// TwinCAT 3 PLC project IoT_HTTP_REST_API
// ProgramVersion: 3.1.4023.0
// libraries:
//   Tc2_EtherCAT, * (Beckhoff Automation GmbH)
//   Tc2_MDP, * (Beckhoff Automation GmbH)
//   Tc2_ModbusSrv, * (Beckhoff Automation GmbH)
//   Tc2_Standard, * (Beckhoff Automation GmbH)
//   Tc2_System, * (Beckhoff Automation GmbH)
//   Tc2_Utilities, * (Beckhoff Automation GmbH)
//   Tc3_IotBase, * (Beckhoff Automation GmbH)
//   Tc3_IPCDiag, * (Beckhoff Automation GmbH)
//   Tc3_JsonXml, * (Beckhoff Automation GmbH)
//   Tc3_Module, * (Beckhoff Automation GmbH)
//   BASIC,3.31,OSCAT
//   VisuSymbols,3.5.10.0,System
// project tree:
//   / Class Diagram.TcCD (not stored), GlobalTextList.TcGTLO (not stored), PlcTask_10ms.TcTTO (not stored), PlcTask_500us.TcTTO (not stored), Task_1ms.TcTTO (not stored), Visualization Manager.TcVMO (not stored)
//   DUTs/ AirValveSimSignals.TcDUT (not stored), ElectrDataModbusTCP.TcDUT (not stored), ElectrDataEthCAT.TcDUT (not stored)
//   DUTs/DataModels/ DriveState_DataModel.TcDUT (not stored), ElectrDevicePeriodicOper_DataModel.TcDUT (not stored), ElectrDeviceContOper_DataModel.TcDUT (not stored), SingleSensor_DataModel.TcDUT (not stored), SingleState_DataModel.TcDUT (not stored), VibAccelarationDataModel.TcDUT (not stored)
//   DUTs/MES/ Order.TcDUT
//   GVLs/ GVL_const.TcGVL, GVL_SW.TcGVL (not stored), GVL_HW.TcGVL (not stored), GVL_Visu.TcGVL (not stored)
//   POUs/EL3443/EL3443/DUTs/ E_EL3443_Phase.TcDUT (not stored), E_EL3443_Total.TcDUT (not stored), ST_EL3443_MUX_REAL.TcDUT (not stored), ST_EL3443_MUX_ULINT.TcDUT (not stored), ST_EL3443_StatusLx.TcDUT (not stored), ST_EL3443_StatusTotal.TcDUT (not stored), ST_EL3443_VariantLx.TcDUT (not stored), ST_EL3443_VariantTotal.TcDUT (not stored), ST_EL3443_VariantValues.TcDUT (not stored)
//   POUs/EL3443/EL3443/ FB_EL3443.TcPOU (not stored)
//   POUs/EL3443/EL3443_DPM/DUTs/ E_EL3443_DPM_Phase.TcDUT (not stored), E_EL3443_DPM_Total.TcDUT (not stored), ST_EL3443_DPM_MUX_REAL.TcDUT (not stored), ST_EL3443_DPM_MUX_ULINT.TcDUT (not stored), ST_EL3443_DPM_StatusLx.TcDUT (not stored), ST_EL3443_DPM_StatusTotal.TcDUT (not stored), ST_EL3443_DPM_VariantLx.TcDUT (not stored), ST_EL3443_DPM_VariantTotal.TcDUT (not stored), ST_EL3443_DPM_VariantValues.TcDUT (not stored)
//   POUs/EL3443/EL3443_DPM/ FB_EL3443_DPM.TcPOU (not stored)
//   POUs/FB/Generic/ CheckLineProducing.TcPOU (not stored), PartsPerMinHistorical.TcPOU (not stored), PartsPerMinInstant.TcPOU (not stored), PartsPerMinInstant2.TcPOU (not stored), ReadMemoryUsage.TcPOU (not stored), TONR.TcPOU (not stored), UnixTimestamp.TcPOU (not stored), ValueChangeDetector.TcPOU (not stored), Valve_Signal_Sim.TcPOU (not stored)
//   POUs/FB/HTTP_REST_API/ HttpGet.TcPOU, ElectricalDevicePeriodicOper.TcPOU, ElectricalDeviceContOper.TcPOU, GenericSensor.TcPOU, GenericState.TcPOU, HttpPost.TcPOU, VibrationSensor.TcPOU
//   POUs/FB/ModbusTCP/ ReadMBSentron_PAC1200.TcPOU (not stored)
//   POUs/FC/ AI_Scale.TcPOU (not stored)
//   POUs/PRG_10ms/ PRG_06_ElectricalMonitoring.TcPOU, PRG_05_ElectricalAnalytics.TcPOU, PRG_01_MAIN.TcPOU, PRG_09_PlcDiagnostic.TcPOU, PRG_08_ProductionStatistics.TcPOU, PRG_10_TempHumidAnalytics.TcPOU, PRG_11_AirFlowAnalytics.TcPOU, PRG_12_OilContaminationAnalytics.TcPOU, PRG_13_MES.TcPOU, Simulation.TcPOU, PRG_02_DataMapping.TcPOU (not stored), PRG_07_LineState.TcPOU, PRG_03_VibrationAnalytics.TcPOU
//   POUs/PRG_1ms/ Main_T1ms.TcPOU (not stored), TimeStamp.TcPOU (not stored)
//   POUs/PRG_500us/ Main_500us.TcPOU (not stored)
//   VISU/ TextList1.TcTLO (not stored), Visualization1.TcVIS (not stored)
// real-time tasks:
//   TASK PlcTask_10ms: cycle T#10ms, priority 20, ADS port 350
//   TASK Task_1ms: cycle T#1ms, priority 1, ADS port 351
//   TASK ProfiNET: cycle T#2ms, priority 2, ADS port 301
//   TASK PlcTask_500us: cycle T#500us, priority 23, ADS port 354
// I/O:
//   DEVICE Device1 (Profinet Device) (disabled), AmsNetId 192.168.149.130.2.1
//     profinet-io-device [Beckhoff Automation TwinCAT PLC PROFINET I/O Device with I/Os, V2.32, 1 port diagnostic supported TwinCAT PN Device]
//       modules: Term 1 (DAP Module), Term 2 (32 Word Output), Term 3 (32 DWord Output), Term 4 (10 Float32 Output), Term 5 (10 Float32 Input)
//   DEVICE Device2 (EtherCAT) (disabled), AmsNetId 192.168.149.130.3.1
//     ElectricalCabinet [EK1100 EtherCAT Coupler (2A E-Bus)]
//       Term_1 (EL3443) [EL3443 3Ch. Power Measuring]
//       Term_2 (EL3443) [EL3443 3Ch. Power Measuring]
//       Term_3 (EL3152) [EL3152 2Ch. Ana Input 4-20mA]
//       Term_4 (EL6601) [EL6601 1 Port Switch (Ethernet, CoE)]
//       Term_99 (EL9011) [EL9011 End Terminal]
//     IO_LinkNode1 (EP6228-0022) [EP6228-0022 (IO Link Master)]
//       modules: Module 1 (DeviceState Inputs Device), Module 2 (DeviceState Inputs), IoLinkNode1_Ch1 (IO-Link Slave), IoLinkNode1_Ch2 (IO-Link Slave), IoLinkNode1_Ch3 (IO-Link Slave), IoLinkNode1_Ch4 (IO-Link Slave), IoLinkNode1_Ch5 (IO-Link Slave), IoLinkNode1_Ch6 (IO-Link Slave), Module 9 (empty), Module 10 (empty)
//     IO_LinkNode2 (EP6224-2022) [EP6224-2022 (IO Link Master)]
//       modules: Module 1 (DeviceState Inputs Device), Module 2 (DeviceState Inputs), IoLinkNode2_Ch1 (IO-Link Slave), IoLinkNode2_Ch2 (IO-Link Slave), IoLinkNode2_Ch3 (IO-Link Slave), IoLinkNode2_Ch4 (IO-Link Slave)
//   DEVICE Device 3 (USB) (disabled)
//     Box 2 (C9900-L100 License-Key-USB-Stick)
// variable links:
//   IoT_HTTP_REST_API/IoT_HTTP_REST_API Instance <-> Device1 (Profinet Device)/profinet-io-device
//     PlcTask_10ms Inputs/GVL_HW.PnIoDevice_10Real_In <-> API/Term 4 (10 Float32 Output)/Subterm 6 (10 Float32 Output)/Inputs/1 Float32 Output[0]
//     PlcTask_10ms Inputs/GVL_HW.PnIoDevice_10Real_In @bit {32..288 step 32} <-> API/Term 4 (10 Float32 Output)/Subterm 6 (10 Float32 Output)/Inputs/1 Float32 Output[{1..9}]  (9 links)
//     PlcTask_10ms Inputs/GVL_HW.PnIoDevice_32DWord_In <-> API/Term 3 (32 DWord Output)/Subterm 5 (32 DWord Output)/Inputs/1 DWord Output[0]
//     PlcTask_10ms Inputs/GVL_HW.PnIoDevice_32DWord_In @bit {32..992 step 32} <-> API/Term 3 (32 DWord Output)/Subterm 5 (32 DWord Output)/Inputs/1 DWord Output[{1..31}]  (31 links)
//     PlcTask_10ms Inputs/GVL_HW.PnIoDevice_32Word_In <-> API/Term 2 (32 Word Output)/Subterm 4 (32 Word Output)/Inputs/1 Word Output[0]
//     PlcTask_10ms Inputs/GVL_HW.PnIoDevice_32Word_In @bit {16..496 step 16} <-> API/Term 2 (32 Word Output)/Subterm 4 (32 Word Output)/Inputs/1 Word Output[{1..31}]  (31 links)
//     PlcTask_10ms Outputs/GVL_HW.PnIoDevice_10Real_Out <-> API/Term 5 (10 Float32 Input)/Subterm 7 (10 Float32 Input)/Outputs/1 Float32 Input[0]
//     PlcTask_10ms Outputs/GVL_HW.PnIoDevice_10Real_Out @bit {32..288 step 32} <-> API/Term 5 (10 Float32 Input)/Subterm 7 (10 Float32 Input)/Outputs/1 Float32 Input[{1..9}]  (9 links)
//   IoT_HTTP_REST_API/IoT_HTTP_REST_API Instance <-> Device2 (EtherCAT)/ElectricalCabinet/Term_1 (EL3443)
//     PlcTask_500us Inputs/Main_500us.ElectricalDevice1.stEL3443_IO.MDP5001_341_Input/MDP5001_341_L1_Basic_Current <-> L1 Basic/Current
//     PlcTask_500us Inputs/Main_500us.ElectricalDevice1.stEL3443_IO.MDP5001_341_Input/MDP5001_341_L2_Basic_Current <-> L2 Basic/Current
//     PlcTask_500us Inputs/Main_500us.ElectricalDevice1.stEL3443_IO.MDP5001_341_Input/MDP5001_341_L3_Basic_Current <-> L3 Basic/Current
//     PlcTask_500us Inputs/Main_500us.ElectricalDevice1.stEL3443_IO.MDP5001_341_Input/MDP5001_341_L1_Basic_Voltage <-> L1 Basic/Voltage
//     PlcTask_500us Inputs/Main_500us.ElectricalDevice1.stEL3443_IO.MDP5001_341_Input/MDP5001_341_L2_Basic_Voltage <-> L2 Basic/Voltage
//     PlcTask_500us Inputs/Main_500us.ElectricalDevice1.stEL3443_IO.MDP5001_341_Input/MDP5001_341_L3_Basic_Voltage <-> L3 Basic/Voltage
//     PlcTask_500us Inputs/Main_500us.ElectricalDevice1.stEL3443_IO.MDP5001_341_Input/MDP5001_341_L1_Power_Active_Power <-> L1 Power/Active Power
//     PlcTask_500us Inputs/Main_500us.ElectricalDevice1.stEL3443_IO.MDP5001_341_Input/MDP5001_341_L2_Power_Active_Power <-> L2 Power/Active Power
//     PlcTask_500us Inputs/Main_500us.ElectricalDevice1.stEL3443_IO.MDP5001_341_Input/MDP5001_341_L3_Power_Active_Power <-> L3 Power/Active Power
//     PlcTask_500us Inputs/Main_500us.ElectricalDevice1.stEL3443_IO.MDP5001_341_Input/MDP5001_341_L1_Power_Apparent_Power <-> L1 Power/Apparent Power
//     PlcTask_500us Inputs/Main_500us.ElectricalDevice1.stEL3443_IO.MDP5001_341_Input/MDP5001_341_L2_Power_Apparent_Power <-> L2 Power/Apparent Power
//     PlcTask_500us Inputs/Main_500us.ElectricalDevice1.stEL3443_IO.MDP5001_341_Input/MDP5001_341_L3_Power_Apparent_Power <-> L3 Power/Apparent Power
//     PlcTask_500us Inputs/Main_500us.ElectricalDevice1.stEL3443_IO.MDP5001_341_Input/MDP5001_341_L1_Power_Power_Factor <-> L1 Power/Power Factor
//     PlcTask_500us Inputs/Main_500us.ElectricalDevice1.stEL3443_IO.MDP5001_341_Input/MDP5001_341_L2_Power_Power_Factor <-> L2 Power/Power Factor
//     PlcTask_500us Inputs/Main_500us.ElectricalDevice1.stEL3443_IO.MDP5001_341_Input/MDP5001_341_L3_Power_Power_Factor <-> L3 Power/Power Factor
//     PlcTask_500us Inputs/Main_500us.ElectricalDevice1.stEL3443_IO.MDP5001_341_Input/MDP5001_341_L1_Power_Reactive_Power <-> L1 Power/Reactive Power
//     PlcTask_500us Inputs/Main_500us.ElectricalDevice1.stEL3443_IO.MDP5001_341_Input/MDP5001_341_L2_Power_Reactive_Power <-> L2 Power/Reactive Power
//     PlcTask_500us Inputs/Main_500us.ElectricalDevice1.stEL3443_IO.MDP5001_341_Input/MDP5001_341_L3_Power_Reactive_Power <-> L3 Power/Reactive Power
//     PlcTask_500us Inputs/Main_500us.ElectricalDevice1.stEL3443_IO.MDP5001_341_Input/MDP5001_341_L1_Status_Current_Guard_Error <-> L1 Status/Current Guard Error
//     PlcTask_500us Inputs/Main_500us.ElectricalDevice1.stEL3443_IO.MDP5001_341_Input/MDP5001_341_L2_Status_Current_Guard_Error <-> L2 Status/Current Guard Error
//     PlcTask_500us Inputs/Main_500us.ElectricalDevice1.stEL3443_IO.MDP5001_341_Input/MDP5001_341_L3_Status_Current_Guard_Error <-> L3 Status/Current Guard Error
//     PlcTask_500us Inputs/Main_500us.ElectricalDevice1.stEL3443_IO.MDP5001_341_Input/MDP5001_341_L1_Status_Current_Guard_Warning <-> L1 Status/Current Guard Warning
//     PlcTask_500us Inputs/Main_500us.ElectricalDevice1.stEL3443_IO.MDP5001_341_Input/MDP5001_341_L2_Status_Current_Guard_Warning <-> L2 Status/Current Guard Warning
//     PlcTask_500us Inputs/Main_500us.ElectricalDevice1.stEL3443_IO.MDP5001_341_Input/MDP5001_341_L3_Status_Current_Guard_Warning <-> L3 Status/Current Guard Warning
//     PlcTask_500us Inputs/Main_500us.ElectricalDevice1.stEL3443_IO.MDP5001_341_Input/MDP5001_341_L1_Status_Inaccurate_Current <-> L1 Status/Inaccurate Current
//     PlcTask_500us Inputs/Main_500us.ElectricalDevice1.stEL3443_IO.MDP5001_341_Input/MDP5001_341_L2_Status_Inaccurate_Current <-> L2 Status/Inaccurate Current
//     PlcTask_500us Inputs/Main_500us.ElectricalDevice1.stEL3443_IO.MDP5001_341_Input/MDP5001_341_L3_Status_Inaccurate_Current <-> L3 Status/Inaccurate Current
//     PlcTask_500us Inputs/Main_500us.ElectricalDevice1.stEL3443_IO.MDP5001_341_Input/MDP5001_341_L1_Status_Inaccurate_Voltage <-> L1 Status/Inaccurate Voltage
//     PlcTask_500us Inputs/Main_500us.ElectricalDevice1.stEL3443_IO.MDP5001_341_Input/MDP5001_341_L2_Status_Inaccurate_Voltage <-> L2 Status/Inaccurate Voltage
//     PlcTask_500us Inputs/Main_500us.ElectricalDevice1.stEL3443_IO.MDP5001_341_Input/MDP5001_341_L3_Status_Inaccurate_Voltage <-> L3 Status/Inaccurate Voltage
//     PlcTask_500us Inputs/Main_500us.ElectricalDevice1.stEL3443_IO.MDP5001_341_Input/MDP5001_341_L1_Status_Overcurrent <-> L1 Status/Overcurrent
//     PlcTask_500us Inputs/Main_500us.ElectricalDevice1.stEL3443_IO.MDP5001_341_Input/MDP5001_341_L2_Status_Overcurrent <-> L2 Status/Overcurrent
//     PlcTask_500us Inputs/Main_500us.ElectricalDevice1.stEL3443_IO.MDP5001_341_Input/MDP5001_341_L3_Status_Overcurrent <-> L3 Status/Overcurrent
//     PlcTask_500us Inputs/Main_500us.ElectricalDevice1.stEL3443_IO.MDP5001_341_Input/MDP5001_341_L1_Status_Overvoltage <-> L1 Status/Overvoltage
//     PlcTask_500us Inputs/Main_500us.ElectricalDevice1.stEL3443_IO.MDP5001_341_Input/MDP5001_341_L2_Status_Overvoltage <-> L2 Status/Overvoltage
//     PlcTask_500us Inputs/Main_500us.ElectricalDevice1.stEL3443_IO.MDP5001_341_Input/MDP5001_341_L3_Status_Overvoltage <-> L3 Status/Overvoltage
//     PlcTask_500us Inputs/Main_500us.ElectricalDevice1.stEL3443_IO.MDP5001_341_Input/MDP5001_341_L1_Status_TxPDO_Toggle <-> L1 Status/TxPDO Toggle
//     PlcTask_500us Inputs/Main_500us.ElectricalDevice1.stEL3443_IO.MDP5001_341_Input/MDP5001_341_L2_Status_TxPDO_Toggle <-> L2 Status/TxPDO Toggle
//     PlcTask_500us Inputs/Main_500us.ElectricalDevice1.stEL3443_IO.MDP5001_341_Input/MDP5001_341_L3_Status_TxPDO_Toggle <-> L3 Status/TxPDO Toggle
//     PlcTask_500us Inputs/Main_500us.ElectricalDevice1.stEL3443_IO.MDP5001_341_Input/MDP5001_341_L1_Status_Voltage_Guard_Error <-> L1 Status/Voltage Guard Error
//     PlcTask_500us Inputs/Main_500us.ElectricalDevice1.stEL3443_IO.MDP5001_341_Input/MDP5001_341_L2_Status_Voltage_Guard_Error <-> L2 Status/Voltage Guard Error
//     PlcTask_500us Inputs/Main_500us.ElectricalDevice1.stEL3443_IO.MDP5001_341_Input/MDP5001_341_L3_Status_Voltage_Guard_Error <-> L3 Status/Voltage Guard Error
//     PlcTask_500us Inputs/Main_500us.ElectricalDevice1.stEL3443_IO.MDP5001_341_Input/MDP5001_341_L1_Status_Voltage_Guard_Warning <-> L1 Status/Voltage Guard Warning
//     PlcTask_500us Inputs/Main_500us.ElectricalDevice1.stEL3443_IO.MDP5001_341_Input/MDP5001_341_L2_Status_Voltage_Guard_Warning <-> L2 Status/Voltage Guard Warning
//     PlcTask_500us Inputs/Main_500us.ElectricalDevice1.stEL3443_IO.MDP5001_341_Input/MDP5001_341_L3_Status_Voltage_Guard_Warning <-> L3 Status/Voltage Guard Warning
//     PlcTask_500us Inputs/Main_500us.ElectricalDevice1.stEL3443_IO.MDP5001_341_Input/MDP5001_341_L1_Status_Voltage_Sign_Bit <-> L1 Status/Voltage Sign Bit
//     PlcTask_500us Inputs/Main_500us.ElectricalDevice1.stEL3443_IO.MDP5001_341_Input/MDP5001_341_L2_Status_Voltage_Sign_Bit <-> L2 Status/Voltage Sign Bit
//     PlcTask_500us Inputs/Main_500us.ElectricalDevice1.stEL3443_IO.MDP5001_341_Input/MDP5001_341_L3_Status_Voltage_Sign_Bit <-> L3 Status/Voltage Sign Bit
//     PlcTask_500us Inputs/Main_500us.ElectricalDevice1.stEL3443_IO.MDP5001_341_Input/MDP5001_341_L1_Timing_Voltage_Last_Zero_Crossing <-> L1 Timing/Voltage Last Zero Crossing
//     PlcTask_500us Inputs/Main_500us.ElectricalDevice1.stEL3443_IO.MDP5001_341_Input/MDP5001_341_L2_Timing_Voltage_Last_Zero_Crossing <-> L2 Timing/Voltage Last Zero Crossing
//     PlcTask_500us Inputs/Main_500us.ElectricalDevice1.stEL3443_IO.MDP5001_341_Input/MDP5001_341_L3_Timing_Voltage_Last_Zero_Crossing <-> L3 Timing/Voltage Last Zero Crossing
//     PlcTask_500us Inputs/Main_500us.ElectricalDevice1.stEL3443_IO.MDP5001_341_Input/MDP5001_341_Total_Basic_Calculated_Neutral_Line_Current <-> Total Basic/Calculated Neutral Line Current
//     PlcTask_500us Inputs/Main_500us.ElectricalDevice1.stEL3443_IO.MDP5001_341_Input/MDP5001_341_Total_Basic_Frequency <-> Total Basic/Frequency
//     PlcTask_500us Inputs/Main_500us.ElectricalDevice1.stEL3443_IO.MDP5001_341_Input/MDP5001_341_Total_Basic_Power_Factor <-> Total Basic/Power Factor
//     PlcTask_500us Inputs/Main_500us.ElectricalDevice1.stEL3443_IO.MDP5001_341_Input/MDP5001_341_Total_Status_Active_Power_Guard_Error <-> Total Status/Active Power Guard Error
//     PlcTask_500us Inputs/Main_500us.ElectricalDevice1.stEL3443_IO.MDP5001_341_Input/MDP5001_341_Total_Status_Active_Power_Guard_Warning <-> Total Status/Active Power Guard Warning
//     PlcTask_500us Inputs/Main_500us.ElectricalDevice1.stEL3443_IO.MDP5001_341_Input/MDP5001_341_Total_Status_Apparent_Power_Guard_Error <-> Total Status/Apparent Power Guard Error
//     PlcTask_500us Inputs/Main_500us.ElectricalDevice1.stEL3443_IO.MDP5001_341_Input/MDP5001_341_Total_Status_Apparent_Power_Guard_Warning <-> Total Status/Apparent Power Guard Warning
//     PlcTask_500us Inputs/Main_500us.ElectricalDevice1.stEL3443_IO.MDP5001_341_Input/MDP5001_341_Total_Status_Frequency_Guard_Error <-> Total Status/Frequency Guard Error
//     PlcTask_500us Inputs/Main_500us.ElectricalDevice1.stEL3443_IO.MDP5001_341_Input/MDP5001_341_Total_Status_Frequency_Guard_Warning <-> Total Status/Frequency Guard Warning
//     PlcTask_500us Inputs/Main_500us.ElectricalDevice1.stEL3443_IO.MDP5001_341_Input/MDP5001_341_Total_Status_Grid_Direction <-> Total Status/Grid Direction
//     PlcTask_500us Inputs/Main_500us.ElectricalDevice1.stEL3443_IO.MDP5001_341_Input/MDP5001_341_Total_Status_Neutral_Current_Guard_Error <-> Total Status/Neutral Current Guard Error
//     PlcTask_500us Inputs/Main_500us.ElectricalDevice1.stEL3443_IO.MDP5001_341_Input/MDP5001_341_Total_Status_Neutral_Current_Guard_Warning <-> Total Status/Neutral Current Guard Warning
//     PlcTask_500us Inputs/Main_500us.ElectricalDevice1.stEL3443_IO.MDP5001_341_Input/MDP5001_341_Total_Status_Power_Quality_Factor <-> Total Status/Power Quality Factor
//     PlcTask_500us Inputs/Main_500us.ElectricalDevice1.stEL3443_IO.MDP5001_341_Input/MDP5001_341_Total_Status_Power_Quality_Guard_Error <-> Total Status/Power Quality Guard Error
//     PlcTask_500us Inputs/Main_500us.ElectricalDevice1.stEL3443_IO.MDP5001_341_Input/MDP5001_341_Total_Status_Power_Quality_Guard_Warning <-> Total Status/Power Quality Guard Warning
//     PlcTask_500us Inputs/Main_500us.ElectricalDevice1.stEL3443_IO.MDP5001_341_Input/MDP5001_341_Total_Status_System_State <-> Total Status/System State
//     PlcTask_500us Inputs/Main_500us.ElectricalDevice1.stEL3443_IO.MDP5001_341_Input/MDP5001_341_Total_Status_TxPDO_State <-> Total Status/TxPDO State
//     PlcTask_500us Inputs/Main_500us.ElectricalDevice1.stEL3443_IO.MDP5001_341_Input/MDP5001_341_Total_Status_TxPDO_Toggle <-> Total Status/TxPDO Toggle
//     PlcTask_500us Inputs/Main_500us.ElectricalDevice1.stEL3443_IO.MDP5001_341_Input/MDP5001_341_Total_Variant_Value_In_Index_1_REAL <-> Total Variant Value In/Index 1 REAL
//     PlcTask_500us Inputs/Main_500us.ElectricalDevice1.stEL3443_IO.MDP5001_341_Input/MDP5001_341_Total_Variant_Value_In_Index_2_REAL <-> Total Variant Value In/Index 2 REAL
//     PlcTask_500us Inputs/Main_500us.ElectricalDevice1.stEL3443_IO.MDP5001_341_Input/MDP5001_341_Total_Variant_Value_In_Index_3_REAL <-> Total Variant Value In/Index 3 REAL
//     PlcTask_500us Inputs/Main_500us.ElectricalDevice1.stEL3443_IO.MDP5001_341_Input/MDP5001_341_Total_Variant_Value_In_Index_4_ULINT <-> Total Variant Value In/Index 4 ULINT
//     PlcTask_500us Inputs/Main_500us.ElectricalDevice1.stEL3443_IO.MDP5001_341_Input/MDP5001_341_Total_Variant_Value_In_TxPDO_Toggle <-> Total Variant Value In/TxPDO Toggle
//     PlcTask_500us Inputs/Main_500us.ElectricalDevice1.stEL3443_IO.MDP5001_341_Input/MDP5001_341_Total_Variant_Value_In_Value_1_REAL <-> Total Variant Value In/Value 1 REAL
//     PlcTask_500us Inputs/Main_500us.ElectricalDevice1.stEL3443_IO.MDP5001_341_Input/MDP5001_341_Total_Variant_Value_In_Value_2_REAL <-> Total Variant Value In/Value 2 REAL
//     PlcTask_500us Inputs/Main_500us.ElectricalDevice1.stEL3443_IO.MDP5001_341_Input/MDP5001_341_Total_Variant_Value_In_Value_3_REAL <-> Total Variant Value In/Value 3 REAL
//     PlcTask_500us Inputs/Main_500us.ElectricalDevice1.stEL3443_IO.MDP5001_341_Input/MDP5001_341_Total_Variant_Value_In_Value_4_ULINT <-> Total Variant Value In/Value 4 ULINT
//     PlcTask_500us Outputs/Main_500us.ElectricalDevice1.stEL3443_IO.MDP5001_341_Output/MDP5001_341_Total_Variant_Value_Out_Index_1_REAL <-> Total Variant Value Out/Index 1 REAL
//     PlcTask_500us Outputs/Main_500us.ElectricalDevice1.stEL3443_IO.MDP5001_341_Output/MDP5001_341_Total_Variant_Value_Out_Index_2_REAL <-> Total Variant Value Out/Index 2 REAL
//     PlcTask_500us Outputs/Main_500us.ElectricalDevice1.stEL3443_IO.MDP5001_341_Output/MDP5001_341_Total_Variant_Value_Out_Index_3_REAL <-> Total Variant Value Out/Index 3 REAL
//     PlcTask_500us Outputs/Main_500us.ElectricalDevice1.stEL3443_IO.MDP5001_341_Output/MDP5001_341_Total_Variant_Value_Out_Index_4_ULINT <-> Total Variant Value Out/Index 4 ULINT
//   IoT_HTTP_REST_API/IoT_HTTP_REST_API Instance <-> Device2 (EtherCAT)/ElectricalCabinet/Term_2 (EL3443)
//     PlcTask_500us Inputs/Main_500us.ElectricalDevice2.stEL3443_IO.MDP5001_341_Input/MDP5001_341_L1_Basic_Current <-> L1 Basic/Current
//     PlcTask_500us Inputs/Main_500us.ElectricalDevice2.stEL3443_IO.MDP5001_341_Input/MDP5001_341_L2_Basic_Current <-> L2 Basic/Current
//     PlcTask_500us Inputs/Main_500us.ElectricalDevice2.stEL3443_IO.MDP5001_341_Input/MDP5001_341_L3_Basic_Current <-> L3 Basic/Current
//     PlcTask_500us Inputs/Main_500us.ElectricalDevice2.stEL3443_IO.MDP5001_341_Input/MDP5001_341_L1_Basic_Voltage <-> L1 Basic/Voltage
//     PlcTask_500us Inputs/Main_500us.ElectricalDevice2.stEL3443_IO.MDP5001_341_Input/MDP5001_341_L2_Basic_Voltage <-> L2 Basic/Voltage
//     PlcTask_500us Inputs/Main_500us.ElectricalDevice2.stEL3443_IO.MDP5001_341_Input/MDP5001_341_L3_Basic_Voltage <-> L3 Basic/Voltage
//     PlcTask_500us Inputs/Main_500us.ElectricalDevice2.stEL3443_IO.MDP5001_341_Input/MDP5001_341_L1_Power_Active_Power <-> L1 Power/Active Power
//     PlcTask_500us Inputs/Main_500us.ElectricalDevice2.stEL3443_IO.MDP5001_341_Input/MDP5001_341_L2_Power_Active_Power <-> L2 Power/Active Power
//     PlcTask_500us Inputs/Main_500us.ElectricalDevice2.stEL3443_IO.MDP5001_341_Input/MDP5001_341_L3_Power_Active_Power <-> L3 Power/Active Power
//     PlcTask_500us Inputs/Main_500us.ElectricalDevice2.stEL3443_IO.MDP5001_341_Input/MDP5001_341_L1_Power_Apparent_Power <-> L1 Power/Apparent Power
//     PlcTask_500us Inputs/Main_500us.ElectricalDevice2.stEL3443_IO.MDP5001_341_Input/MDP5001_341_L2_Power_Apparent_Power <-> L2 Power/Apparent Power
//     PlcTask_500us Inputs/Main_500us.ElectricalDevice2.stEL3443_IO.MDP5001_341_Input/MDP5001_341_L3_Power_Apparent_Power <-> L3 Power/Apparent Power
//     PlcTask_500us Inputs/Main_500us.ElectricalDevice2.stEL3443_IO.MDP5001_341_Input/MDP5001_341_L1_Power_Power_Factor <-> L1 Power/Power Factor
//     PlcTask_500us Inputs/Main_500us.ElectricalDevice2.stEL3443_IO.MDP5001_341_Input/MDP5001_341_L2_Power_Power_Factor <-> L2 Power/Power Factor
//     PlcTask_500us Inputs/Main_500us.ElectricalDevice2.stEL3443_IO.MDP5001_341_Input/MDP5001_341_L3_Power_Power_Factor <-> L3 Power/Power Factor
//     PlcTask_500us Inputs/Main_500us.ElectricalDevice2.stEL3443_IO.MDP5001_341_Input/MDP5001_341_L1_Power_Reactive_Power <-> L1 Power/Reactive Power
//     PlcTask_500us Inputs/Main_500us.ElectricalDevice2.stEL3443_IO.MDP5001_341_Input/MDP5001_341_L2_Power_Reactive_Power <-> L2 Power/Reactive Power
//     PlcTask_500us Inputs/Main_500us.ElectricalDevice2.stEL3443_IO.MDP5001_341_Input/MDP5001_341_L3_Power_Reactive_Power <-> L3 Power/Reactive Power
//     PlcTask_500us Inputs/Main_500us.ElectricalDevice2.stEL3443_IO.MDP5001_341_Input/MDP5001_341_L1_Status_Current_Guard_Error <-> L1 Status/Current Guard Error
//     PlcTask_500us Inputs/Main_500us.ElectricalDevice2.stEL3443_IO.MDP5001_341_Input/MDP5001_341_L2_Status_Current_Guard_Error <-> L2 Status/Current Guard Error
//     PlcTask_500us Inputs/Main_500us.ElectricalDevice2.stEL3443_IO.MDP5001_341_Input/MDP5001_341_L3_Status_Current_Guard_Error <-> L3 Status/Current Guard Error
//     PlcTask_500us Inputs/Main_500us.ElectricalDevice2.stEL3443_IO.MDP5001_341_Input/MDP5001_341_L1_Status_Current_Guard_Warning <-> L1 Status/Current Guard Warning
//     PlcTask_500us Inputs/Main_500us.ElectricalDevice2.stEL3443_IO.MDP5001_341_Input/MDP5001_341_L2_Status_Current_Guard_Warning <-> L2 Status/Current Guard Warning
//     PlcTask_500us Inputs/Main_500us.ElectricalDevice2.stEL3443_IO.MDP5001_341_Input/MDP5001_341_L3_Status_Current_Guard_Warning <-> L3 Status/Current Guard Warning
//     PlcTask_500us Inputs/Main_500us.ElectricalDevice2.stEL3443_IO.MDP5001_341_Input/MDP5001_341_L1_Status_Inaccurate_Current <-> L1 Status/Inaccurate Current
//     PlcTask_500us Inputs/Main_500us.ElectricalDevice2.stEL3443_IO.MDP5001_341_Input/MDP5001_341_L2_Status_Inaccurate_Current <-> L2 Status/Inaccurate Current
//     PlcTask_500us Inputs/Main_500us.ElectricalDevice2.stEL3443_IO.MDP5001_341_Input/MDP5001_341_L3_Status_Inaccurate_Current <-> L3 Status/Inaccurate Current
//     PlcTask_500us Inputs/Main_500us.ElectricalDevice2.stEL3443_IO.MDP5001_341_Input/MDP5001_341_L1_Status_Inaccurate_Voltage <-> L1 Status/Inaccurate Voltage
//     PlcTask_500us Inputs/Main_500us.ElectricalDevice2.stEL3443_IO.MDP5001_341_Input/MDP5001_341_L2_Status_Inaccurate_Voltage <-> L2 Status/Inaccurate Voltage
//     PlcTask_500us Inputs/Main_500us.ElectricalDevice2.stEL3443_IO.MDP5001_341_Input/MDP5001_341_L3_Status_Inaccurate_Voltage <-> L3 Status/Inaccurate Voltage
//     PlcTask_500us Inputs/Main_500us.ElectricalDevice2.stEL3443_IO.MDP5001_341_Input/MDP5001_341_L1_Status_Overcurrent <-> L1 Status/Overcurrent
//     PlcTask_500us Inputs/Main_500us.ElectricalDevice2.stEL3443_IO.MDP5001_341_Input/MDP5001_341_L2_Status_Overcurrent <-> L2 Status/Overcurrent
//     PlcTask_500us Inputs/Main_500us.ElectricalDevice2.stEL3443_IO.MDP5001_341_Input/MDP5001_341_L3_Status_Overcurrent <-> L3 Status/Overcurrent
//     PlcTask_500us Inputs/Main_500us.ElectricalDevice2.stEL3443_IO.MDP5001_341_Input/MDP5001_341_L1_Status_Overvoltage <-> L1 Status/Overvoltage
//     PlcTask_500us Inputs/Main_500us.ElectricalDevice2.stEL3443_IO.MDP5001_341_Input/MDP5001_341_L2_Status_Overvoltage <-> L2 Status/Overvoltage
//     PlcTask_500us Inputs/Main_500us.ElectricalDevice2.stEL3443_IO.MDP5001_341_Input/MDP5001_341_L3_Status_Overvoltage <-> L3 Status/Overvoltage
//     PlcTask_500us Inputs/Main_500us.ElectricalDevice2.stEL3443_IO.MDP5001_341_Input/MDP5001_341_L1_Status_TxPDO_Toggle <-> L1 Status/TxPDO Toggle
//     PlcTask_500us Inputs/Main_500us.ElectricalDevice2.stEL3443_IO.MDP5001_341_Input/MDP5001_341_L2_Status_TxPDO_Toggle <-> L2 Status/TxPDO Toggle
//     PlcTask_500us Inputs/Main_500us.ElectricalDevice2.stEL3443_IO.MDP5001_341_Input/MDP5001_341_L3_Status_TxPDO_Toggle <-> L3 Status/TxPDO Toggle
//     PlcTask_500us Inputs/Main_500us.ElectricalDevice2.stEL3443_IO.MDP5001_341_Input/MDP5001_341_L1_Status_Voltage_Guard_Error <-> L1 Status/Voltage Guard Error
//     PlcTask_500us Inputs/Main_500us.ElectricalDevice2.stEL3443_IO.MDP5001_341_Input/MDP5001_341_L2_Status_Voltage_Guard_Error <-> L2 Status/Voltage Guard Error
//     PlcTask_500us Inputs/Main_500us.ElectricalDevice2.stEL3443_IO.MDP5001_341_Input/MDP5001_341_L3_Status_Voltage_Guard_Error <-> L3 Status/Voltage Guard Error
//     PlcTask_500us Inputs/Main_500us.ElectricalDevice2.stEL3443_IO.MDP5001_341_Input/MDP5001_341_L1_Status_Voltage_Guard_Warning <-> L1 Status/Voltage Guard Warning
//     PlcTask_500us Inputs/Main_500us.ElectricalDevice2.stEL3443_IO.MDP5001_341_Input/MDP5001_341_L2_Status_Voltage_Guard_Warning <-> L2 Status/Voltage Guard Warning
//     PlcTask_500us Inputs/Main_500us.ElectricalDevice2.stEL3443_IO.MDP5001_341_Input/MDP5001_341_L3_Status_Voltage_Guard_Warning <-> L3 Status/Voltage Guard Warning
//     PlcTask_500us Inputs/Main_500us.ElectricalDevice2.stEL3443_IO.MDP5001_341_Input/MDP5001_341_L1_Status_Voltage_Sign_Bit <-> L1 Status/Voltage Sign Bit
//     PlcTask_500us Inputs/Main_500us.ElectricalDevice2.stEL3443_IO.MDP5001_341_Input/MDP5001_341_L2_Status_Voltage_Sign_Bit <-> L2 Status/Voltage Sign Bit
//     PlcTask_500us Inputs/Main_500us.ElectricalDevice2.stEL3443_IO.MDP5001_341_Input/MDP5001_341_L3_Status_Voltage_Sign_Bit <-> L3 Status/Voltage Sign Bit
//     PlcTask_500us Inputs/Main_500us.ElectricalDevice2.stEL3443_IO.MDP5001_341_Input/MDP5001_341_L1_Timing_Voltage_Last_Zero_Crossing <-> L1 Timing/Voltage Last Zero Crossing
//     PlcTask_500us Inputs/Main_500us.ElectricalDevice2.stEL3443_IO.MDP5001_341_Input/MDP5001_341_L2_Timing_Voltage_Last_Zero_Crossing <-> L2 Timing/Voltage Last Zero Crossing
//     PlcTask_500us Inputs/Main_500us.ElectricalDevice2.stEL3443_IO.MDP5001_341_Input/MDP5001_341_L3_Timing_Voltage_Last_Zero_Crossing <-> L3 Timing/Voltage Last Zero Crossing
//     PlcTask_500us Inputs/Main_500us.ElectricalDevice2.stEL3443_IO.MDP5001_341_Input/MDP5001_341_Total_Basic_Calculated_Neutral_Line_Current <-> Total Basic/Calculated Neutral Line Current
//     PlcTask_500us Inputs/Main_500us.ElectricalDevice2.stEL3443_IO.MDP5001_341_Input/MDP5001_341_Total_Basic_Frequency <-> Total Basic/Frequency
//     PlcTask_500us Inputs/Main_500us.ElectricalDevice2.stEL3443_IO.MDP5001_341_Input/MDP5001_341_Total_Basic_Power_Factor <-> Total Basic/Power Factor
//     PlcTask_500us Inputs/Main_500us.ElectricalDevice2.stEL3443_IO.MDP5001_341_Input/MDP5001_341_Total_Status_Active_Power_Guard_Error <-> Total Status/Active Power Guard Error
//     PlcTask_500us Inputs/Main_500us.ElectricalDevice2.stEL3443_IO.MDP5001_341_Input/MDP5001_341_Total_Status_Active_Power_Guard_Warning <-> Total Status/Active Power Guard Warning
//     PlcTask_500us Inputs/Main_500us.ElectricalDevice2.stEL3443_IO.MDP5001_341_Input/MDP5001_341_Total_Status_Apparent_Power_Guard_Error <-> Total Status/Apparent Power Guard Error
//     PlcTask_500us Inputs/Main_500us.ElectricalDevice2.stEL3443_IO.MDP5001_341_Input/MDP5001_341_Total_Status_Apparent_Power_Guard_Warning <-> Total Status/Apparent Power Guard Warning
//     PlcTask_500us Inputs/Main_500us.ElectricalDevice2.stEL3443_IO.MDP5001_341_Input/MDP5001_341_Total_Status_Frequency_Guard_Error <-> Total Status/Frequency Guard Error
//     PlcTask_500us Inputs/Main_500us.ElectricalDevice2.stEL3443_IO.MDP5001_341_Input/MDP5001_341_Total_Status_Frequency_Guard_Warning <-> Total Status/Frequency Guard Warning
//     PlcTask_500us Inputs/Main_500us.ElectricalDevice2.stEL3443_IO.MDP5001_341_Input/MDP5001_341_Total_Status_Grid_Direction <-> Total Status/Grid Direction
//     PlcTask_500us Inputs/Main_500us.ElectricalDevice2.stEL3443_IO.MDP5001_341_Input/MDP5001_341_Total_Status_Neutral_Current_Guard_Error <-> Total Status/Neutral Current Guard Error
//     PlcTask_500us Inputs/Main_500us.ElectricalDevice2.stEL3443_IO.MDP5001_341_Input/MDP5001_341_Total_Status_Neutral_Current_Guard_Warning <-> Total Status/Neutral Current Guard Warning
//     PlcTask_500us Inputs/Main_500us.ElectricalDevice2.stEL3443_IO.MDP5001_341_Input/MDP5001_341_Total_Status_Power_Quality_Factor <-> Total Status/Power Quality Factor
//     PlcTask_500us Inputs/Main_500us.ElectricalDevice2.stEL3443_IO.MDP5001_341_Input/MDP5001_341_Total_Status_Power_Quality_Guard_Error <-> Total Status/Power Quality Guard Error
//     PlcTask_500us Inputs/Main_500us.ElectricalDevice2.stEL3443_IO.MDP5001_341_Input/MDP5001_341_Total_Status_Power_Quality_Guard_Warning <-> Total Status/Power Quality Guard Warning
//     PlcTask_500us Inputs/Main_500us.ElectricalDevice2.stEL3443_IO.MDP5001_341_Input/MDP5001_341_Total_Status_System_State <-> Total Status/System State
//     PlcTask_500us Inputs/Main_500us.ElectricalDevice2.stEL3443_IO.MDP5001_341_Input/MDP5001_341_Total_Status_TxPDO_State <-> Total Status/TxPDO State
//     PlcTask_500us Inputs/Main_500us.ElectricalDevice2.stEL3443_IO.MDP5001_341_Input/MDP5001_341_Total_Status_TxPDO_Toggle <-> Total Status/TxPDO Toggle
//     PlcTask_500us Inputs/Main_500us.ElectricalDevice2.stEL3443_IO.MDP5001_341_Input/MDP5001_341_Total_Variant_Value_In_Index_1_REAL <-> Total Variant Value In/Index 1 REAL
//     PlcTask_500us Inputs/Main_500us.ElectricalDevice2.stEL3443_IO.MDP5001_341_Input/MDP5001_341_Total_Variant_Value_In_Index_2_REAL <-> Total Variant Value In/Index 2 REAL
//     PlcTask_500us Inputs/Main_500us.ElectricalDevice2.stEL3443_IO.MDP5001_341_Input/MDP5001_341_Total_Variant_Value_In_Index_3_REAL <-> Total Variant Value In/Index 3 REAL
//     PlcTask_500us Inputs/Main_500us.ElectricalDevice2.stEL3443_IO.MDP5001_341_Input/MDP5001_341_Total_Variant_Value_In_Index_4_ULINT <-> Total Variant Value In/Index 4 ULINT
//     PlcTask_500us Inputs/Main_500us.ElectricalDevice2.stEL3443_IO.MDP5001_341_Input/MDP5001_341_Total_Variant_Value_In_TxPDO_Toggle <-> Total Variant Value In/TxPDO Toggle
//     PlcTask_500us Inputs/Main_500us.ElectricalDevice2.stEL3443_IO.MDP5001_341_Input/MDP5001_341_Total_Variant_Value_In_Value_1_REAL <-> Total Variant Value In/Value 1 REAL
//     PlcTask_500us Inputs/Main_500us.ElectricalDevice2.stEL3443_IO.MDP5001_341_Input/MDP5001_341_Total_Variant_Value_In_Value_2_REAL <-> Total Variant Value In/Value 2 REAL
//     PlcTask_500us Inputs/Main_500us.ElectricalDevice2.stEL3443_IO.MDP5001_341_Input/MDP5001_341_Total_Variant_Value_In_Value_3_REAL <-> Total Variant Value In/Value 3 REAL
//     PlcTask_500us Inputs/Main_500us.ElectricalDevice2.stEL3443_IO.MDP5001_341_Input/MDP5001_341_Total_Variant_Value_In_Value_4_ULINT <-> Total Variant Value In/Value 4 ULINT
//     PlcTask_500us Outputs/Main_500us.ElectricalDevice2.stEL3443_IO.MDP5001_341_Output/MDP5001_341_Total_Variant_Value_Out_Index_1_REAL <-> Total Variant Value Out/Index 1 REAL
//     PlcTask_500us Outputs/Main_500us.ElectricalDevice2.stEL3443_IO.MDP5001_341_Output/MDP5001_341_Total_Variant_Value_Out_Index_2_REAL <-> Total Variant Value Out/Index 2 REAL
//     PlcTask_500us Outputs/Main_500us.ElectricalDevice2.stEL3443_IO.MDP5001_341_Output/MDP5001_341_Total_Variant_Value_Out_Index_3_REAL <-> Total Variant Value Out/Index 3 REAL
//     PlcTask_500us Outputs/Main_500us.ElectricalDevice2.stEL3443_IO.MDP5001_341_Output/MDP5001_341_Total_Variant_Value_Out_Index_4_ULINT <-> Total Variant Value Out/Index 4 ULINT
//   IoT_HTTP_REST_API/IoT_HTTP_REST_API Instance <-> Device2 (EtherCAT)/IO_LinkNode1 (EP6228-0022)
//     PlcTask_10ms Inputs/GVL_HW.IoLinkNode1Ch{1..6}_SensorTemp <-> IoLinkNode1_Ch{1..6} (IO-Link Slave)/IO-Link Port{1..6}/Contact Temperature Contact Temperature  (6 links)
//     PlcTask_10ms Inputs/GVL_HW.IoLinkNode1Ch{1..6}_VibAccelRmsX <-> IoLinkNode1_Ch{1..6} (IO-Link Slave)/IO-Link Port{1..6}/Vibration Acceleration RMS a-RMS X  (6 links)
//     PlcTask_10ms Inputs/GVL_HW.IoLinkNode1Ch{1..6}_VibAccelRmsY <-> IoLinkNode1_Ch{1..6} (IO-Link Slave)/IO-Link Port{1..6}/Vibration Acceleration RMS a-RMS Y  (6 links)
//     PlcTask_10ms Inputs/GVL_HW.IoLinkNode1Ch{1..6}_VibAccelRmsZ <-> IoLinkNode1_Ch{1..6} (IO-Link Slave)/IO-Link Port{1..6}/Vibration Acceleration RMS a-RMS Z  (6 links)
//   IoT_HTTP_REST_API/IoT_HTTP_REST_API Instance <-> Device2 (EtherCAT)/IO_LinkNode2 (EP6224-2022)
//     PlcTask_10ms Inputs/GVL_HW.IoLinkNode2Ch2_Humidity[1] <-> IoLinkNode2_Ch2 (IO-Link Slave)/IO-Link Port2/Port2: process data[3]
//     PlcTask_10ms Inputs/GVL_HW.IoLinkNode2Ch2_Humidity[2] <-> IoLinkNode2_Ch2 (IO-Link Slave)/IO-Link Port2/Port2: process data[4]
//     PlcTask_10ms Inputs/GVL_HW.IoLinkNode2Ch2_Temperature[1] <-> IoLinkNode2_Ch2 (IO-Link Slave)/IO-Link Port2/Port2: process data[0]
//     PlcTask_10ms Inputs/GVL_HW.IoLinkNode2Ch2_Temperature[2] <-> IoLinkNode2_Ch2 (IO-Link Slave)/IO-Link Port2/Port2: process data[1]
//     PlcTask_10ms Inputs/GVL_HW.IoLinkNode2Ch3_Level <-> IoLinkNode2_Ch3 (IO-Link Slave)/IO-Link Port3/Level
//     PlcTask_10ms Inputs/GVL_HW.IoLinkNode2Ch4_DiffPress <-> IoLinkNode2_Ch4 (IO-Link Slave)/IO-Link Port4/Pressure

// ---- DUTs/MES/Order.TcDUT
TYPE Order :
STRUCT
	id				:	INT;
	LineName		:	STRING(50);
	OrderNo			:	INT;
	OrderState		:	STRING(50);
END_STRUCT
END_TYPE

// ---- GVLs/GVL_const.TcGVL
{attribute 'qualified_only'}
VAR_GLOBAL
		
	HttpServerIpAddress		: STRING		:= '192.168.1.103';
	HttpServerPort			: UINT			:= 8000;
	UserName				: STRING		:= 'TODO';
	Password				: STRING		:= 'TODO';
	
	LineName 				: STRING		:= 'IoT_Industrial';
	MachineName 			: STRING		:= 'device01';
	
	// PLC diagnostic states
	PlcCpuMemUsage			: STRING		:= 'PlcCpuMemoryUsage';
	PlcCpuCore2Usage		: STRING		:= 'PlcCpuCore2Usage';
	PlcCpuCore3Usage		: STRING		:= 'PlcCpuCore3Usage';
	PlcCpuCore2Jitter		: STRING		:= 'PlcCpuCore2Jitter';
	PlcCpuCore3Jitter		: STRING		:= 'PlcCpuCore3Jitter';
	
	// air flow sensor
	AirFlowSensor			: STRING		:= 'AirFlow1';
	AirPresSensor			: STRING		:= 'AirPressure1';
	AirTempSensor			: STRING		:= 'AirTemperature1';
	
	// ambient temperature & humidity sensor
	AmbientTempSensor		: STRING		:= 'AmbientTemperature';
	AmbientHumiditySensor 	: STRING		:= 'AmbientHumidity';


	// vibration sensors 
	VibSensor1 			:STRING			:= 'Vib1';			
	VibSensor2 			:STRING			:= 'Vib2';			
	VibSensor3 			:STRING			:= 'Vib3';			
	VibSensor4 			:STRING			:= 'Vib4';		
	VibSensor5 			:STRING			:= 'Vib5';			
	VibSensor6 			:STRING			:= 'Vib6';		
	
	// air valves
	AirValve1			:STRING			:= 'AirValve1';
	AirValve2			:STRING			:= 'AirValve2';
	AirValve3			:STRING			:= 'AirValve3';
	AirValve4			:STRING			:= 'AirValve4';
	
	// electrical devices  - periodic operation - (motors/drives)
	ElecDevice1 		: STRING 		:= 'ElecDevice1';
	ElecDevice2 		: STRING 		:= 'ElecDevice2';
	
	// electrical devices  - continous operation 
	ElecDevice3 		: STRING 		:= 'ElecDevice3';
	
	DiffPressSensor1	: STRING		:= 'DiffPressSensor1';
	
END_VAR

// ---- POUs/FB/HTTP_REST_API/HttpGet.TcPOU
FUNCTION_BLOCK HttpGet
VAR_INPUT
	HostAddress				: STRING;
	HostPort				: UINT;

	// REST API endpoint
	ApiEndpoint				: STRING(255);
	
	// HTTP GET Command
	HttpGetCmd				: BOOL;
END_VAR

VAR
	bStart 				: BOOL;
	SetParameter		: BOOL:=TRUE;
	
	nSuccess			: UDINT;	
	nFails				: UDINT;

	HttpResponse		: STRING(5000);
	nHttpState			: UDINT; 
	
	fbIotHttpClient		: FB_IotHttpClient;
	URI					: STRING(255);
												
	fbIotHttpRequest	: FB_IotHttpRequest;
	fbJsonDomParser		: FB_JsonDomParser;
	JsonHttpResponse	: SJsonValue;
	
	JsonMessageMember01	: SJsonValue;
	JsonMessageMember02	: SJsonValue;
	JsonMessageMember03	: SJsonValue;

	State				: UDINT;
	idx					: UDINT;

END_VAR
VAR_OUTPUT
	Error				: BOOL;
	HttpResponseState	: UDINT;			// HTTP response state code
	
	OrderID				: STRING(255);
	OrderNo				: INT;
	ProductKey			: STRING(255);
END_VAR

(*
This FB creates HTTP GET request and gets JsonPayload as body from ApiEndpoint.
*)

IF SetParameter THEN
	SetParameter := FALSE;
	fbIotHttpClient.sHostName:=   HostAddress;
	fbIotHttpClient.nHostPort:= HostPort;
	fbIotHttpClient.bKeepAlive := TRUE;
	fbIotHttpClient.tConnectionTimeout := T#10S;
END_IF

IF HttpGetCmd  THEN
	HttpGetCmd := FALSE;
	Error := FALSE;
	State := 10;
END_IF

fbIotHttpClient.Execute();

CASE State OF

	10: // CREATE HTTP REQUEST
		URI := ApiEndpoint;
		IF fbIotHttpRequest.SendRequest(sUri := URI,
										fbClient 		:= fbIotHttpClient,
										eRequestType 	:= ETcIotHttpRequestType.HTTP_Get,
										pContent 		:= 0,
										nContentSize 	:= 0,
										fbHeader 		:= 0)
		THEN
			State := 20;	
		END_IF
	
		
	20: // GET HTTP RESPONSE
		IF NOT fbIotHttpRequest.bBusy THEN
			IF NOT fbIotHttpRequest.bError THEN
					HttpResponseState 	:= fbIotHttpRequest.nStatusCode;
					fbIotHttpRequest.GetContent(pContent := ADR(HttpResponse),
								nContentSize := SIZEOF(HttpResponse),
								bSetNullTermination := TRUE);
								
					IF fbIotHttpRequest.nStatusCode >=200 AND fbIotHttpRequest.nStatusCode < 300 THEN
						nSuccess 	:= nSuccess + 1;
						State 		:= 30;
					END_IF
			ELSE
				// error handling
				nFails 		:= nFails + 1;
				State 		:= 0;
			END_IF
		END_IF

		
	30: // HANDLE RESPONSE
		JsonHttpResponse := fbIotHttpRequest.GetJsonDomContent(fbJsonDomParser);
		IF JsonHttpResponse <> 0 THEN
			
			JsonMessageMember01 := fbJsonDomParser.FindMember(JsonHttpResponse,'id');
			OrderID := fbJsonDomParser.GetString(JsonMessageMember01);
			
			JsonMessageMember02 := fbJsonDomParser.FindMember(JsonHttpResponse,'order_no');
			OrderNo := DINT_TO_INT(fbJsonDomParser.GetInt(JsonMessageMember02));
			
			
			JsonMessageMember03 := fbJsonDomParser.FindMember(JsonHttpResponse,'product_key');
			ProductKey := fbJsonDomParser.GetString(JsonMessageMember03);
				
		END_IF
		State := 0;
	
END_CASE

END_FUNCTION_BLOCK

// ---- POUs/FB/HTTP_REST_API/ElectricalDevicePeriodicOper.TcPOU
FUNCTION_BLOCK ElectricalDevicePeriodicOper
VAR_INPUT
	LineName					: STRING(40);
	MachineName 				: STRING(40);
	DeviceName					: STRING(40);
	TimeStamp					: ULINT;
	DeviceElectricalData 		: ElectrDataEthCAT;
	DeviceRunning				: BOOL;
	SynchPulse					: BOOL;
	Enable						: BOOL;
END_VAR
VAR_OUTPUT
	// REST API Endpoint
	ApiEndpoint 					: STRING(255);
	
	// HTTP body as JSON payload
	JsonPayload 				: STRING(4000);
	
	// HTTP POST Command
	HttpPostCmd 				: BOOL;
END_VAR
VAR
	SetParameter 				: BOOL := TRUE;
		
	// state machine
	nState						: INT;		
		
	// JSON document
  	fbJson			: FB_JsonSaxWriter;
	fbJsonDataType	: FB_JsonReadWriteDataType;
	stValues		: ElectrDevicePeriodicOper_DataModel;	
	
	// device state detection
	rtrigDeviceRunning: R_TRIG;
	ftrigDeviceRunning: F_TRIG;

	// device state
	DeviceState			: BOOL;

	// safety watchdog
	tonWatchdog : TON;	
	
	StoppingCntr 	: INT;
	StoppedCntr 	: INT;
	
	 // Drive States
     RunningState	: BOOL := FALSE;
     StoppingState	: BOOL := FALSE;
     StoppedState	: BOOL := FALSE;
	 DriveStates	: DriveState_DataModel; 
END_VAR

(*
This FB evaluates electrical data from EL3443 when electrical device is in 'Running'
state and creates input data (API Endpoint and JSON body) for HTTP POST request.
*)

IF Enable THEN
		DeviceState := DeviceRunning;
		
		// synchronisation pulse from FB input
		stValues.SynchPulse := SynchPulse;
		
		// edge detection for drive state evaluation
		rtrigDeviceRunning(CLK:=DeviceState);	
		ftrigDeviceRunning(CLK:=DeviceState);	
		
		IF SetParameter THEN
			SetParameter := FALSE;
			HttpPostCmd := FALSE;
			
			// create mqtt topic
			ApiEndpoint := 'electrical-device-periodic-operation';
			
			// constant entry in json payload
			stValues.LineName := LineName;
			stValues.MachineName := MachineName;
			stValues.DeviceName := DeviceName;
		END_IF
		
		
		// evaluate device state
		CASE nState OF
		0:
		// IDLE
			StoppingCntr 		:= 0;
			StoppedCntr 		:= 0;
			RunningState 		:= FALSE;
			StoppingState	 	:= FALSE;
			StoppedState 		:= FALSE;
			HttpPostCmd  		:= FALSE;
			stValues.DeviceState := DriveStates.StoppedState;
			
			IF rtrigDeviceRunning.Q THEN
				// sequence watchdog
				tonWatchdog.IN := TRUE; 
				nState := 10;
			END_IF
			
		10:
		// RUNNING
			RunningState := TRUE;
			stValues.DeviceState := DriveStates.RunningState;
			
			HttpPostCmd := TRUE;
			
			IF ftrigDeviceRunning.Q THEN
				RunningState := FALSE;
				nState := 20;
			END_IF
		
		20:
		// STOPPING
			StoppingState 			:= TRUE;
			stValues.DeviceState 	:= DriveStates.StoppingState;
			tonWatchdog.IN := FALSE;
			
			IF StoppingState THEN StoppingCntr := StoppingCntr + 1; END_IF
			
			IF StoppingCntr = 3 THEN
				StoppingState := FALSE;
				nState := 30;
			END_IF
		
		30:
		// STOPPED
			StoppedState 			:= TRUE;
			stValues.DeviceState 	:= DriveStates.StoppedState;
		
			IF StoppedState THEN StoppedCntr := StoppedCntr + 1; END_IF
			
			IF StoppedCntr = 2 THEN
				StoppedState := FALSE;
				HttpPostCmd := FALSE;
				nState := 0;
			END_IF
			
		END_CASE
		
		
		IF HttpPostCmd THEN
			//write electrical data from FB input to JSON payload
			stValues.ElectricalData := DeviceElectricalData;
			stValues.TimeStamp := TimeStamp;
		
			//create JSON message
			fbJson.ResetDocument();
			fbJsonDataType.AddJsonValueFromSymbol(fbJson, 
												  'ElectrDevicePeriodicOper_DataModel',
												  SIZEOF(stValues),
												  ADR(stValues));
			fbJson.CopyDocument(JsonPayload, SIZEOF(JsonPayload));
		END_IF
ELSE
		HttpPostCmd := FALSE;
		tonWatchdog.IN := FALSE;
		nState := 0;
END_IF

IF tonWatchdog.ET > T#10S THEN
	nState := 0;
END_IF
tonWatchdog(PT:=T#10S);

END_FUNCTION_BLOCK

// ---- POUs/FB/HTTP_REST_API/ElectricalDeviceContOper.TcPOU
FUNCTION_BLOCK ElectricalDeviceContOper
VAR_INPUT
	LineName					: STRING(40);
	MachineName 				: STRING(40);
	DeviceName					: STRING(40);
	TimeStamp					: ULINT;
	DeviceElectricalData 		: ElectrDataModbusTCP;
	Enable						: BOOL;
END_VAR
VAR_OUTPUT
	// REST API Endpoint
	ApiEndpoint 			: STRING(255);
	
	// HTTP body as JSON payload
	JsonPayload 			: STRING(4000);
	
	// HTTP POST Command
	HttpPostCmd 			: BOOL;
END_VAR
VAR
	SetParameter 			: BOOL := TRUE;		
		
	// JSON document
  	fbJson			: FB_JsonSaxWriter;
	fbJsonDataType	: FB_JsonReadWriteDataType;
	stValues		: ElectrDeviceContOper_DataModel;	
		
END_VAR

(*
This FB evaluates continously  electrical data from Sentron 7KT PAC1200
and creates input data (API Endpoint and JSON body) for HTTP POST request
*)

IF Enable THEN	
		
		IF SetParameter THEN
			SetParameter := FALSE;
			HttpPostCmd := FALSE;
			// create REST API endpoint
			ApiEndpoint := 'electrical-device-continous-operation';
			
			// constant entry in json payload
			stValues.LineName := LineName;
			stValues.MachineName := MachineName;
			stValues.DeviceName := DeviceName;
		END_IF
		
		stValues.TimeStamp := TimeStamp;
		stValues.ElectricalData := DeviceElectricalData;
		
		//create JSON message
		fbJson.ResetDocument();
		fbJsonDataType.AddJsonValueFromSymbol(fbJson, 
												'ElectrDeviceContOper_DataModel', 
												SIZEOF(stValues), 
												ADR(stValues));
		fbJson.CopyDocument(JsonPayload, SIZEOF(JsonPayload));
		
		HttpPostCmd := TRUE;
ELSE
		HttpPostCmd := FALSE;
END_IF

END_FUNCTION_BLOCK

// ---- POUs/FB/HTTP_REST_API/GenericSensor.TcPOU
FUNCTION_BLOCK GenericSensor
VAR_INPUT
	LineName	: STRING(40);
	MachineName : STRING(40);
	SensorName	: STRING(40);
	TimeStamp	: ULINT;
	Value		: REAL;	 
	Enable		: BOOL; //enable sensor evaluation
END_VAR
VAR_OUTPUT
	// REST API Endpoint
	ApiEndpoint 	: STRING(255);
	
	// HTTP body as JSON payload
	JsonPayload		: STRING(4000);
	
	// HTTP POST Command
	HttpPostCmd 	: BOOL;
END_VAR
VAR
	SetParameter : BOOL := TRUE;

	stValues		: SingleSensor_DataModel;	
	
	// JSON document
  	fbJson			: FB_JsonSaxWriter;
	fbJsonDataType	: FB_JsonReadWriteDataType;
	
	// safety watchdog
	tonWatchdog : TON;
END_VAR

(*
This FB evaluates analog value and creates input data (API Endpoint and JSON body) for HTTP POST request 
*) 

IF Enable THEN
	
	IF SetParameter THEN
		SetParameter := FALSE;
		// create REST API endpoint
		ApiEndpoint := '/generic-sensor';
		
		// constant entry in json payload
		stValues.LineName := LineName;
		stValues.MachineName := MachineName;
		stValues.SensorName := SensorName;
	END_IF
	
	stValues.timeStamp := TimeStamp;
	stValues.SensorValue := Value;
		
	// create JSON message
	
	fbJson.ResetDocument();
	fbJsonDataType.AddJsonValueFromSymbol(fbJson, 'SingleSensor_DataModel', SIZEOF(stValues), ADR(stValues));
	fbJson.CopyDocument(JsonPayload, SIZEOF(JsonPayload));
	
	HttpPostCmd := TRUE;
ELSE
	HttpPostCmd := FALSE;
END_IF;

END_FUNCTION_BLOCK

// ---- POUs/FB/HTTP_REST_API/GenericState.TcPOU
FUNCTION_BLOCK GenericState
VAR_INPUT
	LineName	: STRING(40);
	MachineName : STRING(40);
	StateName	: STRING(40);
	TimeStamp	: ULINT;
	Value		: INT;	 
	Enable		: BOOL; 		//enable state evaluation
END_VAR
VAR_OUTPUT
	// REST API Endpoint
	ApiEndpoint 	: STRING(255);
	
	// HTTP body as JSON payload
	JsonPayload		: STRING(4000);
	
	// HTTP POST Command
	HttpPostCmd 	: BOOL;
END_VAR
VAR
	SetParameter : BOOL := TRUE;

	stValues		: SingleState_DataModel;	
	
	// JSON document
  	fbJson			: FB_JsonSaxWriter;
	fbJsonDataType	: FB_JsonReadWriteDataType;
		

	// temporary mqtt topic
	TopicString : STRING;
	
	// safety watchdog
	tonWatchdog : TON;
END_VAR

(*
This FB evaluates single state and creates input data (API Endpoint and JSON body) for HTTP POST request 
*) 

IF Enable THEN
	
	IF SetParameter THEN
		SetParameter := FALSE;
		// create REST API endpoint
		ApiEndpoint := '/generic-state';

		// constant entry in json payload
		stValues.LineName := LineName;
		stValues.MachineName := MachineName;
		stValues.StateName := StateName;
	END_IF
	
	stValues.TimeStamp := TimeStamp;
	stValues.StateValue := Value;
		
	// create JSON message
	fbJson.ResetDocument();
	fbJsonDataType.AddJsonValueFromSymbol(fbJson, 'SingleState_DataModel', SIZEOF(stValues), ADR(stValues));
	fbJson.CopyDocument(JsonPayload, SIZEOF(JsonPayload));
		
	HttpPostCmd := TRUE;
ELSE
	HttpPostCmd := FALSE;
END_IF;

END_FUNCTION_BLOCK

// ---- POUs/FB/HTTP_REST_API/HttpPost.TcPOU
FUNCTION_BLOCK HttpPost
VAR_INPUT

	HostAddress				: STRING;
	HostPort				: UINT;
	
	// Creditials 
	UserName				: STRING;
	UserPassword			: STRING;
	
	// REST API endpoint
	ApiEndpoint				: STRING(255);
	
	// JSON 
	JsonPayload				: STRING(4000);
	
	// HTTP POST Command
	HttpPostCmd				: BOOL;
END_VAR
VAR
	HeaderAdded			: BOOL;
	SetParameter		: BOOL:=TRUE;
	State				: UDINT;
	
	Success				: UDINT;	
	Fails				: UDINT;
	
	
	URI							: STRING(255);
	
	fbIotHttpClient				: FB_IotHttpClient;											
	fbIotHttpHeaderFieldMap		: FB_IotHttpHeaderFieldMap;	 // header
	fbIotHttpRequest			: FB_IotHttpRequest;
	fbJsonDomParser				: FB_JsonDomParser;
	fbJsonBody					: FB_JsonDomParser;
	
	
	HttpResponse				: STRING(5000);
	JsonHttpResponse			: SJsonValue;
	JsonMessageMember			: SJsonValue;
	
	message						: STRING(255);
END_VAR

VAR_OUTPUT
	Error						: BOOL;
	HttpResponseState			: UDINT;
END_VAR

(*
This FB creates HTTP POST request and sends JsonPayload as body to ApiEndpoint.
*)

IF SetParameter THEN
	SetParameter := FALSE;
	fbIotHttpClient.sHostName:=   HostAddress;
	fbIotHttpClient.nHostPort:= HostPort;
	fbIotHttpClient.bKeepAlive := TRUE;
	fbIotHttpClient.tConnectionTimeout := T#10S;
	
	IF NOT HeaderAdded THEN
		fbIotHttpHeaderFieldMap.AddField('Content-Type', 'application/json', FALSE);
		
	END_IF
END_IF


IF HttpPostCmd  THEN
	HttpPostCmd := FALSE;
	Error := FALSE;
	State := 10;
END_IF

fbIotHttpClient.Execute();

CASE State OF

	10: // CREATE REQUEST 
		URI := ApiEndpoint;
		fbJsonBody.ParseDocument(JsonPayload);
		
		IF fbIotHttpRequest.SendJsonDomRequest(sUri := URI,
										fbClient 		:= fbIotHttpClient,
										eRequestType 	:= ETcIotHttpRequestType.HTTP_POST,
										fbJson			:= fbJsonBody,
										fbHeader 		:= fbIotHttpHeaderFieldMap)
		THEN
			State := 11;	
		END_IF
		
	11: // GET RESPONSE
		IF NOT fbIotHttpRequest.bBusy THEN
			HttpResponseState 		:= fbIotHttpRequest.nStatusCode;
			fbIotHttpRequest.GetContent(pContent := ADR(HttpResponse),
										nContentSize := SIZEOF(HttpResponse),
										bSetNullTermination := TRUE);
			IF fbIotHttpRequest.bError THEN
				Error 		:= TRUE;
				// HANDLE ERROR HERE //
				Fails 		:= Fails + 1;
				State 		:= 0;
			ELSE
				Error 		:= FALSE;
				Success 	:= Success + 1;
				State 		:= 12;
			END_IF
		END_IF

	12: // HANDLE RESPONSE
		JsonHttpResponse := fbIotHttpRequest.GetJsonDomContent(fbJsonDomParser);
		IF JsonHttpResponse <> 0 THEN
			JsonMessageMember := fbJsonDomParser.FindMember(JsonHttpResponse,'Message');
			message := fbJsonDomParser.GetString(JsonMessageMember);
		END_IF
		State := 0;
END_CASE;

END_FUNCTION_BLOCK

// ---- POUs/FB/HTTP_REST_API/VibrationSensor.TcPOU
FUNCTION_BLOCK VibrationSensor
VAR_INPUT
	LineName			: STRING(40);
	MachineName 		: STRING(40);
	SensorName			: STRING(40);
	TimeStamp			: ULINT;
	VibAccelX			: REAL;
    VibAccelY			: REAL;
    VibAccelZ			: REAL;	
    SensorTemperature	: REAL;
	MotorState			: BOOL;	
	Enable				: BOOL;
END_VAR
VAR_OUTPUT
	// REST API Endpoint
	ApiEndpoint 	: STRING(255);
	
	// HTTP body as JSON payload
	JsonPayload		: STRING(4000);
	
	// HTTP POST Command
	HttpPostCmd 	: BOOL;
END_VAR
VAR
	SetParameter 		: BOOL := TRUE;
	
	// state machine
	nState				: INT := 0;
	
	// JSON document
  	fbJson				: FB_JsonSaxWriter;
	fbJsonDataType		: FB_JsonReadWriteDataType;
	sJsonDocument		: STRING(4000);
	stValues			: VibAccelarationDataModel;	
		
	// temporary mqtt topic
	TopicString 		: STRING;

	// motor status 
	rtrigMotorState		: R_TRIG;
	ftrigMotorState		: F_TRIG;
	 
	// safety watchdog
	tonWatchdog 		: TON;
	
	StoppingCntr 		: INT;
	StoppedCntr 		: INT;
	
	 //Motor state
	 StartingState		: BOOL := FALSE;
     RunningState		: BOOL := FALSE;
     StoppingState		: BOOL := FALSE;
     StoppedState		: BOOL := FALSE;
	 DriveStates		: DriveState_DataModel; 
	
END_VAR

(*
This FB calculates analytics when motor status is TRUE.

During this state vibration's values from axis x,y,z of the sensor
are accumulated and data (API Endpoint and JSON body) for HTTP POST request will be created at falling
edge of the motor state.

Vibration sensor needs to be located ar the motor or its gearing/coupling 
*)

IF SetParameter THEN
	SetParameter := FALSE;
	// create REST API endpoint
	ApiEndpoint := '/vibration-sensor';
	
	// constant entry in json payload
	stValues.LineName := LineName;
	stValues.MachineName := MachineName;
	stValues.SensorName := SensorName;
END_IF

// detect motor state (running/stopped)
rtrigMotorState(CLK:=MotorState);
ftrigMotorState(CLK:=MotorState);

IF ENABLE THEN
	CASE nState OF
	0:
		ClearData();
		
		IF rtrigMotorState.Q THEN
			tonWatchdog.IN := TRUE;
			nState := 10;
		END_IF
		
	10:
	// RUNNING
		RunningState := TRUE;
		stValues.TimeStamp := TimeStamp;
		stValues.VibAccelTotRmsX := stValues.VibAccelTotRmsX + VibAccelX;
		stValues.VibAccelTotRmsY := stValues.VibAccelTotRmsY + VibAccelY;
		stValues.VibAccelTotRmsZ := stValues.VibAccelTotRmsZ + VibAccelZ;
		stValues.SensorTemperature := SensorTemperature;
	
		IF ftrigMotorState.Q THEN
			RunningState := FALSE;
			nState := 20;
		END_IF
	
	20:
	// STOPPING
		StoppingState := TRUE;
		stValues.TimeStamp := TimeStamp;
		stValues.VibAccelTotRmsX := stValues.VibAccelTotRmsX + VibAccelX;
		stValues.VibAccelTotRmsY := stValues.VibAccelTotRmsY + VibAccelY;
		stValues.VibAccelTotRmsZ := stValues.VibAccelTotRmsZ + VibAccelZ;
		stValues.SensorTemperature := SensorTemperature;
		
		StoppingCntr := StoppingCntr + 1;
		
		IF StoppingCntr = 2 THEN
			StoppingState := FALSE;
			nState := 30;
		END_IF
	
	30:
	// STOPPED
		StoppedState := TRUE;
		stValues.TimeStamp := TimeStamp;
		stValues.VibAccelTotRmsX := ROUND(stValues.VibAccelTotRmsX + VibAccelX, 4);
		stValues.VibAccelTotRmsY := ROUND(stValues.VibAccelTotRmsY + VibAccelY, 4);
		stValues.VibAccelTotRmsZ := ROUND(stValues.VibAccelTotRmsZ + VibAccelZ, 4);
		stValues.SensorTemperature := ROUND(SensorTemperature, 2);
		
		//create JSON message
		
		fbJson.ResetDocument();
		fbJsonDataType.AddJsonValueFromSymbol(fbJson, 'VibAccelarationDataModel', SIZEOF(stValues), ADR(stValues));
		fbJson.CopyDocument(JsonPayload, SIZEOF(JsonPayload));
		
	
		StoppedCntr := StoppedCntr + 1;
		
		IF StoppedCntr = 2 THEN
			StoppedState := FALSE;
			HttpPostCmd := TRUE;
			nState := 0;
		END_IF
		
		tonWatchdog.IN := FALSE;
		
	END_CASE
	
	//Watchdog 7 seconds, restart of sequence
	IF tonWatchdog.ET > T#7S AND nState <> 0 THEN
		nState := 0;
	END_IF
ELSE
	tonWatchdog.IN := FALSE;
	ClearData();
END_IF

	tonWatchdog(PT:=T#10S);

METHOD ClearData
VAR_INPUT
END_VAR
nState			:= 0;
StoppingCntr 	:= 0;
StoppedCntr 	:= 0;
RunningState 	:= FALSE;
StoppingState 	:= FALSE;
StoppedState 	:= FALSE;
stValues.VibAccelTotRmsX := 0.0;
stValues.VibAccelTotRmsY := 0.0;
stValues.VibAccelTotRmsZ := 0.0;

HttpPostCmd := FALSE;
END_METHOD

END_FUNCTION_BLOCK

// ---- POUs/PRG_10ms/PRG_06_ElectricalMonitoring.TcPOU
PROGRAM PRG_06_ElectricalMonitoring
VAR
	ElectDeviceContOper					: ElectricalDeviceContOper;
	ElectDeviceContOperPostHttp			: HttpPost;
	ElectrDeviceContOper				: ReadMBSentron_PAC1200;
END_VAR

ElectDeviceContOper(
    LineName := GVL_const.LineName,
    MachineName := GVL_const.MachineName,
    DeviceName := GVL_const.ElecDevice3,
    TimeStamp := GVL_SW.Unix_TimeStamp,
    DeviceElectricalData := ElectrDeviceContOper.ElectricalData,
    Enable := GVL_Visu.LineRunning); // ElectricalDeviceContOper
ElectDeviceContOperPostHttp(
    HostAddress := GVL_const.HttpServerIpAddress,
    HostPort := GVL_const.HttpServerPort,
    ApiEndpoint := ElectDeviceContOper.ApiEndpoint,
    JsonPayload := ElectDeviceContOper.JsonPayload,
    HttpPostCmd := ElectDeviceContOper.HttpPostCmd); // HttpPost
// Read electrical data over Modbus TCP from Sentron 7KT PAC1200 and send it continously by MQTT.
// IP address of Sentron device
ElectrDeviceContOper(IpAddress := '192.168.1.177', RequestTime := T#100MS, Enable := GVL_Visu.LineRunning); // ReadMBSentron_PAC1200

END_PROGRAM

// ---- POUs/PRG_10ms/PRG_05_ElectricalAnalytics.TcPOU
PROGRAM PRG_05_ElectricalAnalytics
VAR
	ElectricalDevice				: ARRAY[1..2] OF ElectricalDevicePeriodicOper;
	ElectricalDevicePostHttp		: ARRAY[1..2] OF HttpPost;
		
	SyncPulseElecDevice1: TP;
	SyncPulseElecDevice2: TP;

END_VAR
VAR // added by the converter: edge detectors and wires of the graphical bodies
    _s1, _s2 : ElectrDataEthCAT;
END_VAR


// PAGE Electrical Motor1 ---
// Read electrical data from EL3443 module and send  it by MQTT during device RUN state.
// It allows analytics of periodically switched device
// compose _s1 : ElectrDataEthCAT
_s1.ActPowerTot := Main_500us.ElectricalDevice1.stVariantValues.stTotal.fPtot;
_s1.ReactPowerTot := Main_500us.ElectricalDevice1.stVariantValues.stTotal.fQtot;
_s1.ApparPowerTot := Main_500us.ElectricalDevice1.stVariantValues.stTotal.fStot;
_s1.PowerFact := Main_500us.ElectricalDevice1.stVariantValues.stTotal.fPower_Factor;
_s1.PQF := Main_500us.ElectricalDevice1.stVariantValues.stTotal.fPQF;
_s1.ActPowerL1 := Main_500us.ActPowL1ElecDevice1;
_s1.ReactPowerL1 := Main_500us.ReactPowL1ElecDevice1;
_s1.ApparPowerL1 := Main_500us.AppPowL1ElecDevice1;
_s1.CurrentL1 := GVL_Visu.ElCurrentL1[1];
_s1.VoltL1 := Main_500us.VoltL1ElecDevice1;
_s1.PowFactL1 := Main_500us.PowFactL1ElecDevice1;
_s1.VoltL1_THD := Main_500us.ElectricalDevice1.stVariantValues.astLx[1].fTHD_U;
_s1.CurrentL1_THD := Main_500us.ElectricalDevice1.stVariantValues.astLx[1].fTHD_I;
_s1.CurrentL1_harm := Main_500us.ElectricalDevice1.stVariantValues.astLx[1].fHarmonics_I;
_s1.ActPowerL2 := Main_500us.ActPowL2ElecDevice1;
_s1.ReactPowerL2 := Main_500us.ReactPowL2ElecDevice1;
_s1.ApparPowerL2 := Main_500us.AppPowL2ElecDevice1;
_s1.CurrentL2 := GVL_Visu.ElCurrentL2[1];
_s1.VoltL2 := Main_500us.VoltL2ElecDevice1;
_s1.PowFactL2 := Main_500us.PowFactL2ElecDevice1;
_s1.VoltL2_THD := Main_500us.ElectricalDevice1.stVariantValues.astLx[2].fTHD_U;
_s1.CurrentL2_THD := Main_500us.ElectricalDevice1.stVariantValues.astLx[2].fTHD_I;
_s1.CurrentL2_harm := Main_500us.ElectricalDevice1.stVariantValues.astLx[2].fHarmonics_I;
_s1.ActPowerL3 := Main_500us.ActPowL3ElecDevice1;
_s1.ReactPowerL3 := Main_500us.ReactPowL3ElecDevice1;
_s1.ApparPowerL3 := Main_500us.AppPowL3ElecDevice1;
_s1.CurrentL3 := GVL_Visu.ElCurrentL3[1];
_s1.VoltL3 := Main_500us.VoltL3ElecDevice1;
_s1.PowFactL3 := Main_500us.PowFactL3ElecDevice1;
_s1.VoltL3_THD := Main_500us.ElectricalDevice1.stVariantValues.astLx[3].fTHD_U;
_s1.CurrentL3_THD := Main_500us.ElectricalDevice1.stVariantValues.astLx[3].fTHD_I;
_s1.CurrentL3_harm := Main_500us.ElectricalDevice1.stVariantValues.astLx[3].fHarmonics_I;
SyncPulseElecDevice1(IN := GVL_Visu.MotorRunning[1], PT := T#500ms); // TP
ElectricalDevice[1](
    LineName := GVL_const.LineName,
    MachineName := GVL_const.MachineName,
    DeviceName := GVL_const.ElecDevice1,
    TimeStamp := GVL_SW.Unix_TimeStamp,
    DeviceElectricalData := _s1,
    DeviceRunning := GVL_Visu.MotorRunning[1],
    SynchPulse := SyncPulseElecDevice1.Q,
    Enable := GVL_Visu.LineRunning); // ElectricalDevicePeriodicOper
ElectricalDevicePostHttp[1](
    HostAddress := GVL_const.HttpServerIpAddress,
    HostPort := GVL_const.HttpServerPort,
    ApiEndpoint := ElectricalDevice[1].ApiEndpoint,
    JsonPayload := ElectricalDevice[1].JsonPayload,
    HttpPostCmd := ElectricalDevice[1].HttpPostCmd); // HttpPost

// PAGE Electrical Motor2 ---
// compose _s2 : ElectrDataEthCAT
_s2.ActPowerTot := Main_500us.ElectricalDevice2.stVariantValues.stTotal.fPtot;
_s2.ReactPowerTot := Main_500us.ElectricalDevice2.stVariantValues.stTotal.fQtot;
_s2.ApparPowerTot := Main_500us.ElectricalDevice2.stVariantValues.stTotal.fStot;
_s2.PowerFact := Main_500us.ElectricalDevice2.stVariantValues.stTotal.fPower_Factor;
_s2.PQF := Main_500us.ElectricalDevice2.stVariantValues.stTotal.fPQF;
_s2.ActPowerL1 := Main_500us.ActPowL1ElecDevice2;
_s2.ReactPowerL1 := Main_500us.ReactPowL1ElecDevice2;
_s2.ApparPowerL1 := Main_500us.AppPowL1ElecDevice2;
_s2.CurrentL1 := GVL_Visu.ElCurrentL1[2];
_s2.VoltL1 := Main_500us.VoltL1ElecDevice2;
_s2.PowFactL1 := Main_500us.PowFactL1ElecDevice2;
_s2.VoltL1_THD := Main_500us.ElectricalDevice2.stVariantValues.astLx[1].fTHD_U;
_s2.CurrentL1_THD := Main_500us.ElectricalDevice2.stVariantValues.astLx[1].fTHD_I;
_s2.CurrentL1_harm := Main_500us.ElectricalDevice2.stVariantValues.astLx[1].fHarmonics_I;
_s2.ActPowerL2 := Main_500us.ActPowL2ElecDevice2;
_s2.ReactPowerL2 := Main_500us.ReactPowL2ElecDevice2;
_s2.ApparPowerL2 := Main_500us.AppPowL2ElecDevice2;
_s2.CurrentL2 := GVL_Visu.ElCurrentL2[2];
_s2.VoltL2 := Main_500us.VoltL2ElecDevice2;
_s2.PowFactL2 := Main_500us.PowFactL2ElecDevice2;
_s2.VoltL2_THD := Main_500us.ElectricalDevice2.stVariantValues.astLx[2].fTHD_U;
_s2.CurrentL2_THD := Main_500us.ElectricalDevice2.stVariantValues.astLx[2].fTHD_I;
_s2.CurrentL2_harm := Main_500us.ElectricalDevice2.stVariantValues.astLx[2].fHarmonics_I;
_s2.ActPowerL3 := Main_500us.ActPowL3ElecDevice2;
_s2.ReactPowerL3 := Main_500us.ReactPowL3ElecDevice2;
_s2.ApparPowerL3 := Main_500us.AppPowL3ElecDevice2;
_s2.CurrentL3 := GVL_Visu.ElCurrentL3[2];
_s2.VoltL3 := Main_500us.VoltL3ElecDevice2;
_s2.PowFactL3 := Main_500us.PowFactL3ElecDevice2;
_s2.VoltL3_THD := Main_500us.ElectricalDevice2.stVariantValues.astLx[3].fTHD_U;
_s2.CurrentL3_THD := Main_500us.ElectricalDevice2.stVariantValues.astLx[3].fTHD_I;
_s2.CurrentL3_harm := Main_500us.ElectricalDevice2.stVariantValues.astLx[3].fHarmonics_I;
SyncPulseElecDevice2(IN := GVL_Visu.MotorRunning[2], PT := T#500ms); // TP
// Read electrical data from EL3443 module and send  it by MQTT during device RUN state.
// It allows analytics of periodically switched device
ElectricalDevice[2](
    lineName := GVL_const.LineName,
    machineName := GVL_const.MachineName,
    DeviceName := GVL_const.ElecDevice2,
    TimeStamp := GVL_SW.Unix_TimeStamp,
    DeviceElectricalData := _s2,
    DeviceRunning := GVL_Visu.MotorRunning[2],
    SynchPulse := SyncPulseElecDevice2.Q,
    Enable := GVL_Visu.LineRunning); // ElectricalDevicePeriodicOper
ElectricalDevicePostHttp[2](
    HostAddress := GVL_const.HttpServerIpAddress,
    HostPort := GVL_const.HttpServerPort,
    UserName := GVL_const.UserName,
    UserPassword := GVL_const.Password,
    ApiEndpoint := ElectricalDevice[2].ApiEndpoint,
    JsonPayload := ElectricalDevice[2].JsonPayload,
    HttpPostCmd := ElectricalDevice[2].HttpPostCmd); // HttpPost
// Main_500us.rCurrL1_BC1: input not connected
// Main_500us.rCurrL2_BC1: input not connected
// Main_500us.rCurrL3_BC1: input not connected
// Main_500us.rCurrL1_BC2: input not connected
// Main_500us.rCurrL2_BC2: input not connected
// Main_500us.rCurrL3_BC2: input not connected

END_PROGRAM

// ---- POUs/PRG_10ms/PRG_01_MAIN.TcPOU
PROGRAM PRG_01_MAIN
VAR
			tonRecycle100ms			:	TON;
			tonRecycle5sec			:	TON;
END_VAR

PRG_02_DataMapping();

Simulation();

PRG_03_VibrationAnalytics();
PRG_07_LineState();
PRG_08_ProductionStatistics();
PRG_09_PlcDiagnostic();

PRG_13_MES();

tonRecycle5sec(IN:=NOT tonRecycle5sec.Q, PT:=T#5S);
tonRecycle100ms(IN:=NOT tonRecycle100ms.Q, PT:=T#500MS);

// 500 ms cycle monitoring
IF tonRecycle100ms.Q THEN
	PRG_11_AirFlowAnalytics();
END_IF

// slow process values monitoring
IF tonRecycle5sec.Q THEN
	PRG_10_TempHumidAnalytics();
	PRG_12_OilContaminationAnalytics();
END_IF

END_PROGRAM

// ---- POUs/PRG_10ms/Simulation.TcPOU
PROGRAM Simulation
VAR
	idx			: BYTE;
	tp1Motor 	: ARRAY[1..6] OF TP;
	tp2Motor 	: ARRAY[1..6] OF TP;
	
	VibSensorBase : ARRAY[1..6] OF REAL := [0.7, 0.2, 0.3, 0.8, 0.5, 0.1];
	VibSensorOffset : ARRAY[1..6] OF REAL;
	
	AirFlowRateBase			:	REAL := 30.0;
	AirPressureBase			:	REAL := 6.0;
	AirTemperatureBase		:	REAL := 20.0;
	
	AirValve				:	ARRAY [1..6] OF Valve_Signal_Sim;
	AirValvePositionSim		: 	ARRAY [1..6] OF INT;
	
	tonProductPos			:	TON;
	rtrigProductSensor		: 	R_TRIG;
	
	tp1AutoMode				:	TP;
	tp2AutoMode				:	TP;
	tp1AutoModeTime			:	TIME := T#5S;
	tp2AutoModeTime			:	TIME := T#2S;
	rtrigAutoMode			:	R_TRIG;

	rndTime1				: INT;
	rndTime2				: INT;
	
	ElecSample1				: INT;
	ElecSample2				: INT;
	ElecCurrentOffsetL1		: REAL;
	ElecCurrentOffsetL2		: REAL;	
	ElecCurrentOffsetL3		: REAL;
	ElCurrentL1Base			: ARRAY[1..2] OF ARRAY[1..100] OF REAL := 
								[
								[0, 0, 0.1, 0.3, 0.45, 0.60, 0.70, 0.80, 0.95, 1.1, 1.3, 1.4, 1.55, 1.6, 1.59,1.55, 
								1.45, 1.3, 1.2, 1.1, 1.05, 1.0, 0.95, 0.9, 0.85, 0.83, 0.80, 0.78, 0.75, 0.74, 0.72,
								0.70, 0.69, 0.69, 0.69, 0.68, 0.68, 0.67, 0.67, 0.65, 0.64, 0.62, 0.60, 0.58, 0.58, 0.57, 0.56, 0.55, 0.55,
								0, 0, 0, 0, 0, 0, 0, 0, 0, 0],
								[0, 0, 0.1, 0.2, 0.3, 0.55, 1.0, 1.3, 1.5, 1.7, 1.8, 1.81, 1.7, 1.5, 1.2, 1.22, 1.19, 1.23,
								1.19, 1.21, 1.18, 1.22, 1.19, 1.23, 1.17, 1.21, 1.20, 1.18, 1.21, 1.18, 1.22, 1.17, 1.23,
								1.19, 1.21, 1.19, 1.20, 1.19, 1.20, 1.19, 1.21, 1.20, 1.20, 1.22, 1.19, 1.21, 1.18, 1.21, 1.2, 1.2,
								1.21, 1.20, 1.20, 1.22, 1.19, 1.21, 1.18, 1.21, 1.2, 1.2, 40(1.2)]];
								
	ElCurrentL2Base			: ARRAY[1..2] OF ARRAY[1..100] OF REAL := 
								[
								[0, 0, 0.1, 0.3, 0.45, 0.60, 0.70, 0.80, 0.95, 1.1, 1.3, 1.4, 1.55, 1.6, 1.59,1.55, 
								1.45, 1.3, 1.2, 1.1, 1.05, 1.0, 0.95, 0.9, 0.85, 0.83, 0.80, 0.78, 0.75, 0.74, 0.72,
								0.70, 0.69, 0.69, 0.69, 0.68, 0.68, 0.67, 0.67, 0.65, 0.64, 0.62, 0.60, 0.58, 0.58, 0.57, 0.56, 0.55, 0.55,
								0, 0, 0, 0, 0, 0, 0, 0, 0, 0],
								[0, 0, 0.1, 0.2, 0.3, 0.55, 1.0, 1.3, 1.5, 1.7, 1.8, 1.81, 1.7, 1.5, 1.2, 1.22, 1.19, 1.23,
								1.19, 1.21, 1.18, 1.22, 1.19, 1.23, 1.17, 1.21, 1.20, 1.18, 1.21, 1.18, 1.22, 1.17, 1.23,
								1.19, 1.21, 1.19, 1.20, 1.19, 1.20, 1.19, 1.21, 1.20, 1.20, 1.22, 1.19, 1.21, 1.18, 1.21, 1.2, 1.2,
								1.21, 1.20, 1.20, 1.22, 1.19, 1.21, 1.18, 1.21, 1.2, 1.2]];

	ElCurrentL3Base			: ARRAY[1..2] OF ARRAY[1..100] OF REAL := 
								[
								[0, 0, 0.1, 0.3, 0.45, 0.60, 0.70, 0.80, 0.95, 1.1, 1.3, 1.4, 1.55, 1.6, 1.59,1.55, 
								1.45, 1.3, 1.2, 1.1, 1.05, 1.0, 0.95, 0.9, 0.85, 0.83, 0.80, 0.78, 0.75, 0.74, 0.72,
								0.70, 0.69, 0.69, 0.69, 0.68, 0.68, 0.67, 0.67, 0.65, 0.64, 0.62, 0.60, 0.58, 0.58, 0.57, 0.56, 0.55, 0.55,
								0, 0, 0, 0, 0, 0, 0, 0, 0, 0],
								[0, 0, 0.1, 0.2, 0.3, 0.55, 1.0, 1.3, 1.5, 1.7, 1.8, 1.81, 1.7, 1.5, 1.2, 1.22, 1.19, 1.23,
								1.19, 1.21, 1.18, 1.22, 1.19, 1.23, 1.17, 1.21, 1.20, 1.18, 1.21, 1.18, 1.22, 1.17, 1.23,
								1.19, 1.21, 1.19, 1.20, 1.19, 1.20, 1.19, 1.21, 1.20, 1.20, 1.22, 1.19, 1.21, 1.18, 1.21, 1.2, 1.2,
								1.21, 1.20, 1.20, 1.22, 1.19, 1.21, 1.18, 1.21, 1.2, 1.2]];
END_VAR

IF GVL_Visu.ButtonStart THEN
	
	GVL_Visu.LineRunning := TRUE;
	// simulate motor running signals
	tp1Motor[1](IN:= NOT tp2Motor[1].Q, PT:= T#1S);
	tp2Motor[1](IN:= NOT tp1Motor[1].Q, PT:= T#500MS);
	
	tp1Motor[2](IN:= NOT tp2Motor[2].Q, PT:= T#2S);
	tp2Motor[2](IN:= NOT tp1Motor[2].Q, PT:= T#300MS);
	
	tp1Motor[3](IN:= NOT tp2Motor[3].Q, PT:= T#1.7S);
	tp2Motor[3](IN:= NOT tp1Motor[3].Q, PT:= T#500MS);
	
	tp1Motor[4](IN:= NOT tp2Motor[4].Q, PT:= T#1S);
	tp2Motor[4](IN:= NOT tp1Motor[4].Q, PT:= T#1S);
	
	tp1Motor[5](IN:= NOT tp2Motor[5].Q, PT:= T#500MS);
	tp2Motor[5](IN:= NOT tp1Motor[5].Q, PT:= T#2S);
	
	tp1Motor[6](IN:= NOT tp2Motor[6].Q, PT:= T#1S);
	tp2Motor[6](IN:= NOT tp1Motor[6].Q, PT:= T#300MS);
	
	// simulate auto/manual mode
	tp1AutoMode(IN:= NOT tp2AutoMode.Q, PT:= tp1AutoModeTime);
	tp2AutoMode(IN:= NOT tp1AutoMode.Q, PT:= tp2AutoModeTime);
	
	rtrigAutoMode(CLK:=tp1AutoMode.Q);
	
	// generate random time windows of auto and manual period  
	IF  rtrigAutoMode.Q THEN
		rndTime1 := RDM2(last:=2, low:=0, high:=70);
		tp1AutoModeTime:=T#5S + INT_TO_TIME(rndTime1*100);
		
		rndTime2 := RDM2(last:=5, low:=0, high:=30);
		tp2AutoModeTime:=T#2S + INT_TO_TIME(rndTime2*100);
	END_IF

	GVL_Visu.AutoMode := tp2AutoMode.Q;
	
	
	// simulate vibration sensors
	FOR idx := 1 TO 6 DO
		GVL_Visu.MotorRunning[idx] := tp1Motor[idx].Q;
		
		GVL_Visu.VibrationSensorX[idx] := VibSensorBase[idx] + RDM(0.4);
		GVL_Visu.VibrationSensorY[idx] := VibSensorBase[idx] + RDM(0.4);
		GVL_Visu.VibrationSensorZ[idx] := VibSensorBase[idx] + RDM(0.4);	
	END_FOR
	
	// simulate air supply sensors
	GVL_Visu.AirFlowRate 		:= AirFlowRateBase + 2* RDM(0.5);
	GVL_Visu.AirPressure		:= AirPressureBase + 2 * RDM(0.9); 
	GVL_Visu.AirTemperature		:= AirTemperatureBase + RDM(0.3);
	
	
	// simulate air valves
	AirValve[1](StartSim			:= TRUE, 
			    ExtendCmdTime		:= T#500MS,
			    ExtendTime 			:= T#1800MS,
			    RetractCmdTime 		:= T#600MS,
			    RetractTime  		:= T#2000MS);
			  
	AirValve[2](StartSim			:= TRUE, 
			    ExtendCmdTime		:= T#50MS,
			    ExtendTime 			:= T#180MS,
			    RetractCmdTime 		:= T#50MS,
			    RetractTime  		:= T#145MS);
				
	AirValve[3](StartSim			:= TRUE, 
			    ExtendCmdTime		:= T#100MS,
			    ExtendTime 			:= T#1200MS,
			    RetractCmdTime 		:= T#120MS,
			    RetractTime  		:= T#1500MS);
				
	AirValve[4](StartSim			:= TRUE, 
			    ExtendCmdTime		:= T#30MS,
			    ExtendTime 			:= T#120MS,
			    RetractCmdTime 		:= T#30MS,
			    RetractTime  		:= T#120MS);
				
	FOR idx := 1 TO 4 DO
		GVL_Visu.AirValve[idx].ExtendCmd := AirValve[idx].ExtendCmd;
		GVL_Visu.AirValve[idx].ExtendFeedback := AirValve[idx].ExtendFeedback;
		GVL_Visu.AirValve[idx].RetractCmd := AirValve[idx].RetractCmd;
		GVL_Visu.AirValve[idx].RetractFeedback := AirValve[idx].RetractFeedback;
		GVL_Visu.AirValvePositionSim[idx] := SEL (NOT GVL_Visu.AirValveEnable[idx], AirValve[idx].nState, 0);
	END_FOR
	
	// simulate product position on the conveyor
	tonProductPos(IN:= NOT tonProductPos.Q, PT:=T#200MS);
	IF tonProductPos.Q THEN
		GVL_Visu.ProductPosition := GVL_Visu.ProductPosition + TO_INT(GVL_Visu.LineSpeed / 5);
	END_IF
	
	IF GVL_Visu.ProductPosition >= 190 THEN
		GVL_Visu.ProductPosition := 0;
	END_IF
	
	// simulate product sensor acitivation
	IF GVL_Visu.ProductPosition >= 175 AND
		 GVL_Visu.ProductPosition <190 THEN
	GVL_Visu.SensorProductActive := TRUE;
	ELSE
		GVL_Visu.SensorProductActive := FALSE;
	END_IF;
	
	// simulate product counting
	rtrigProductSensor(CLK:=GVL_Visu.SensorProductActive);
	IF rtrigProductSensor.Q THEN
		GVL_Visu.OkProductCount := GVL_Visu.OkProductCount + 1;
	END_IF
	
	// simulate electrical current curve of motor 1
	IF GVL_Visu.MotorRunning[1] THEN
		ElecSample1 := ElecSample1+1;
		ElecSample1 := SEL(ElecSample1=60, ElecSample1, 1);
		IF ElecSample1 < 20 OR ElecSample1 > 40 THEN
			ElecCurrentOffsetL1 := RDM(0.67) * 0.05;
			ElecCurrentOffsetL2 := RDM(0.23) * 0.05;
			ElecCurrentOffsetL3 := RDM(0.72) * 0.05;
		ELSE
			ElecCurrentOffsetL1 := RDM(0.31) * 0.05;
			ElecCurrentOffsetL2 := RDM(0.63) * 0.05;
			ElecCurrentOffsetL3 := RDM(0.46) * 0.05;
		END_IF
		GVL_Visu.ElCurrentL1[1] := 	ElCurrentL1Base[1][ElecSample1] + ElecCurrentOffsetL1;
		GVL_Visu.ElCurrentL2[1] := 	ElCurrentL2Base[1][ElecSample1] + ElecCurrentOffsetL2;
		GVL_Visu.ElCurrentL3[1] := 	ElCurrentL3Base[1][ElecSample1] + ElecCurrentOffsetL3;
	ELSE
		ElecSample1 := 0;
		GVL_Visu.ElCurrentL1[1] := 0;
		GVL_Visu.ElCurrentL2[1] := 0;
		GVL_Visu.ElCurrentL3[1] := 0;
	END_IF
	
	// simulate electrical current curve of motor 2
	IF GVL_Visu.MotorRunning[2] THEN
		ElecSample2 := ElecSample2+1;
		ElecSample2 := SEL(ElecSample2=60, ElecSample2, 1);
		GVL_Visu.ElCurrentL1[2] := 	ElCurrentL1Base[2][ElecSample2];
		GVL_Visu.ElCurrentL2[2] := 	ElCurrentL2Base[2][ElecSample2];
		GVL_Visu.ElCurrentL3[2] := 	ElCurrentL3Base[2][ElecSample2];
	ELSE
		ElecSample2 := 0;
		GVL_Visu.ElCurrentL1[2] := 0;
		GVL_Visu.ElCurrentL2[2] := 0;
		GVL_Visu.ElCurrentL3[2] := 0;
	END_IF
	
	// simulate ambient temperature & humidity
	GVL_Visu.AmbientTemperature := 19.0 + 2* RDM(0.7);
	GVL_Visu.AmbientHumidity	:= 60.0 + 3 * RDM(0.5);
	
	// simulate pressure difference for oil contamination sensor
	GVL_Visu.OilDiffPressure := 0.4 + RDM(0.1) * 0.2;
  
ELSE
	GVL_Visu.LineRunning := FALSE;
	tp1AutoMode(IN:=FALSE);
	tp2AutoMode(IN:=FALSE);
	
	GVL_Visu.AutoMode := tp1AutoMode.Q;
	
	FOR idx := 1 TO 4 DO
		AirValve[idx](StartSim := FALSE);
	END_FOR
	
	FOR idx := 1 TO 6 DO
		tp1Motor[idx](IN:= FALSE);
		tp2Motor[idx](IN:= FALSE);	
		GVL_Visu.MotorRunning[idx] := tp1Motor[idx].Q;		
	END_FOR
	
	GVL_Visu.ElCurrentL1[1] := 0;
	GVL_Visu.ElCurrentL2[1] := 0;
	GVL_Visu.ElCurrentL3[1] := 0;
	
	GVL_Visu.ElCurrentL1[2] := 0;
	GVL_Visu.ElCurrentL2[2] := 0;
	GVL_Visu.ElCurrentL3[2] := 0;
	
END_IF

END_PROGRAM

// ---- POUs/PRG_10ms/PRG_03_VibrationAnalytics.TcPOU
PROGRAM PRG_03_VibrationAnalytics
VAR
	VibSensor					: ARRAY [1..6] OF VibrationSensor;
	VibSensorPostHttp			: ARRAY [1..6] OF HttpPost;	
END_VAR


// PAGE Vibration Sensor 1 ----
VibSensor[1](
    LineName := GVL_const.LineName,
    MachineName := GVL_const.MachineName,
    SensorName := GVL_const.VibSensor1,
    TimeStamp := GVL_SW.Unix_TimeStamp,
    VibAccelX := GVL_Visu.VibrationSensorX[1],
    VibAccelY := GVL_Visu.VibrationSensorY[1],
    VibAccelZ := GVL_Visu.VibrationSensorZ[1],
    SensorTemperature := GVL_SW.VibSensor1Temp,
    MotorState := GVL_Visu.MotorRunning[1],
    Enable := GVL_Visu.LineRunning AND GVL_Visu.VibrationSensorsEnable); // VibrationSensor
VibSensorPostHttp[1](
    HostAddress := GVL_const.HttpServerIpAddress,
    HostPort := GVL_const.HttpServerPort,
    ApiEndpoint := VibSensor[1].ApiEndpoint,
    JsonPayload := VibSensor[1].JsonPayload,
    HttpPostCmd := VibSensor[1].HttpPostCmd); // HttpPost

// PAGE Vibration Sensor 2 ---
VibSensor[2](
    LineName := GVL_const.LineName,
    MachineName := GVL_const.MachineName,
    SensorName := GVL_const.VibSensor2,
    TimeStamp := GVL_SW.Unix_TimeStamp,
    VibAccelX := GVL_Visu.VibrationSensorX[2],
    VibAccelY := GVL_Visu.VibrationSensorY[2],
    VibAccelZ := GVL_Visu.VibrationSensorZ[2],
    SensorTemperature := GVL_SW.VibSensor2Temp,
    MotorState := GVL_Visu.MotorRunning[2],
    Enable := GVL_Visu.LineRunning AND GVL_Visu.VibrationSensorsEnable); // VibrationSensor
VibSensorPostHttp[2](
    HostAddress := GVL_const.HttpServerIpAddress,
    HostPort := GVL_const.HttpServerPort,
    ApiEndpoint := VibSensor[2].ApiEndpoint,
    JsonPayload := VibSensor[2].JsonPayload,
    HttpPostCmd := VibSensor[2].HttpPostCmd); // HttpPost

// PAGE Vibration Sensor 3 ---
VibSensor[3](
    LineName := GVL_const.LineName,
    MachineName := GVL_const.MachineName,
    SensorName := GVL_const.VibSensor3,
    TimeStamp := GVL_SW.Unix_TimeStamp,
    VibAccelX := GVL_Visu.VibrationSensorX[3],
    VibAccelY := GVL_Visu.VibrationSensorY[3],
    VibAccelZ := GVL_Visu.VibrationSensorZ[3],
    SensorTemperature := GVL_SW.VibSensor3Temp,
    MotorState := GVL_Visu.MotorRunning[3],
    Enable := GVL_Visu.LineRunning AND GVL_Visu.VibrationSensorsEnable); // VibrationSensor
VibSensorPostHttp[3](
    HostAddress := GVL_const.HttpServerIpAddress,
    HostPort := GVL_const.HttpServerPort,
    ApiEndpoint := VibSensor[3].ApiEndpoint,
    JsonPayload := VibSensor[3].JsonPayload,
    HttpPostCmd := VibSensor[3].HttpPostCmd); // HttpPost

// PAGE Vibration Sensor 4 ---
VibSensor[4](
    LineName := GVL_const.LineName,
    MachineName := GVL_const.MachineName,
    SensorName := GVL_const.VibSensor4,
    TimeStamp := GVL_SW.Unix_TimeStamp,
    VibAccelX := GVL_Visu.VibrationSensorX[4],
    VibAccelY := GVL_Visu.VibrationSensorY[4],
    VibAccelZ := GVL_Visu.VibrationSensorZ[4],
    SensorTemperature := GVL_SW.VibSensor4Temp,
    MotorState := GVL_Visu.MotorRunning[4],
    Enable := GVL_Visu.LineRunning AND GVL_Visu.VibrationSensorsEnable); // VibrationSensor
VibSensorPostHttp[4](
    HostAddress := GVL_const.HttpServerIpAddress,
    HostPort := GVL_const.HttpServerPort,
    ApiEndpoint := VibSensor[4].ApiEndpoint,
    JsonPayload := VibSensor[4].JsonPayload,
    HttpPostCmd := VibSensor[4].HttpPostCmd); // HttpPost

// PAGE Vibration Sensor 5 ---
VibSensor[5](
    LineName := GVL_const.LineName,
    MachineName := GVL_const.MachineName,
    SensorName := GVL_const.VibSensor5,
    TimeStamp := GVL_SW.Unix_TimeStamp,
    VibAccelX := GVL_Visu.VibrationSensorX[5],
    VibAccelY := GVL_Visu.VibrationSensorY[5],
    VibAccelZ := GVL_Visu.VibrationSensorZ[5],
    SensorTemperature := GVL_SW.VibSensor5Temp,
    MotorState := GVL_Visu.MotorRunning[5],
    Enable := GVL_Visu.LineRunning AND GVL_Visu.VibrationSensorsEnable); // VibrationSensor
VibSensorPostHttp[5](
    HostAddress := GVL_const.HttpServerIpAddress,
    HostPort := GVL_const.HttpServerPort,
    ApiEndpoint := VibSensor[5].ApiEndpoint,
    JsonPayload := VibSensor[5].JsonPayload,
    HttpPostCmd := VibSensor[5].HttpPostCmd); // HttpPost

// PAGE Vibration Sensor 6 ---
VibSensor[6](
    LineName := GVL_const.LineName,
    MachineName := GVL_const.MachineName,
    SensorName := GVL_const.VibSensor6,
    TimeStamp := GVL_SW.Unix_TimeStamp,
    VibAccelX := GVL_Visu.VibrationSensorX[6],
    VibAccelY := GVL_Visu.VibrationSensorY[6],
    VibAccelZ := GVL_Visu.VibrationSensorZ[6],
    SensorTemperature := GVL_SW.VibSensor6Temp,
    MotorState := GVL_Visu.MotorRunning[6],
    Enable := GVL_Visu.LineRunning AND GVL_Visu.VibrationSensorsEnable); // VibrationSensor
VibSensorPostHttp[6](
    HostAddress := GVL_const.HttpServerIpAddress,
    HostPort := GVL_const.HttpServerPort,
    ApiEndpoint := VibSensor[6].ApiEndpoint,
    JsonPayload := VibSensor[6].JsonPayload,
    HttpPostCmd := VibSensor[6].HttpPostCmd); // HttpPost
// GVL.BS1_Accel_RMS_X: input not connected
// GVL.BS1_Accel_RMS_Y: input not connected
// GVL.BS1_Accel_RMS_Z: input not connected
// GVL.Drv_RotTable_25N0_M10_RUNNING: input not connected
// GVL.AutoMode: input not connected
// GVL.BS2_Accel_RMS_X: input not connected
// GVL.BS2_Accel_RMS_Y: input not connected
// GVL.BS2_Accel_RMS_Z: input not connected
// GVL.Drv_RotTable_25N0_M10_RUNNING: input not connected
// GVL.AutoMode: input not connected
// GVL.BS3_Accel_RMS_X: input not connected
// GVL.BS3_Accel_RMS_Y: input not connected
// GVL.BS3_Accel_RMS_Z: input not connected
// GVL.Drv_RotTable_25N0_M10_RUNNING: input not connected
// GVL.AutoMode: input not connected
// GVL.BS4_Accel_RMS_X: input not connected
// GVL.BS4_Accel_RMS_Y: input not connected
// GVL.BS4_Accel_RMS_Z: input not connected
// GVL.Drv_RotTable_25N0_M10_RUNNING: input not connected
// GVL.AutoMode: input not connected
// GVL.BS5_Accel_RMS_X: input not connected
// GVL.BS5_Accel_RMS_Y: input not connected
// GVL.BS5_Accel_RMS_Z: input not connected
// GVL.Drv_InfeedBelt2_10N31_M21_RIGHT_RUNNING: input not connected
// GVL.AutoMode: input not connected
// GVL.BS6_Accel_RMS_X: input not connected
// GVL.BS6_Accel_RMS_Y: input not connected
// GVL.BS6_Accel_RMS_Z: input not connected
// GVL.Drv_InfeedBelt2_10N31_M21_RIGHT_RUNNING: input not connected
// GVL.AutoMode: input not connected

END_PROGRAM

// ---- POUs/PRG_10ms/PRG_07_LineState.TcPOU
PROGRAM PRG_07_LineState
VAR
	CheckLine1Producing: CheckLineProducing;
	
	ValueChangeDetector	:	ARRAY[1..6] OF ValueChangeDetector;
	GenericState		:	ARRAY[1..6] OF GenericState;
	PostHttp			:	ARRAY[1..6] OF HttpPost;
	tpValueChangeDelay	:	ARRAY[1..6] OF TP;
	
END_VAR


// PAGE Check if line is producing --
CheckLine1Producing(OkProductNumber := GVL_Visu.OkProductCount); // CheckLineProducing
GVL_Visu.LineProducing := CheckLine1Producing.LineProducing;

// PAGE Send line states over MQTT ---
PostHttp[1](
    HostAddress := GVL_const.HttpServerIpAddress,
    HostPort := GVL_const.HttpServerPort,
    ApiEndpoint := GenericState[1].ApiEndpoint,
    JsonPayload := GenericState[1].JsonPayload,
    HttpPostCmd := GenericState[1].HttpPostCmd); // HttpPost
PostHttp[2](
    HostAddress := GVL_const.HttpServerIpAddress,
    HostPort := GVL_const.HttpServerPort,
    ApiEndpoint := GenericState[2].ApiEndpoint,
    JsonPayload := GenericState[2].JsonPayload,
    HttpPostCmd := GenericState[2].HttpPostCmd); // HttpPost
ValueChangeDetector[1](Value := BOOL_TO_INT(GVL_Visu.AutoMode)); // ValueChangeDetector
tpValueChangeDelay[1](IN := ValueChangeDetector[1].ValueChanged, PT := T#50MS); // TP
GenericState[1](
    LineName := GVL_const.LineName,
    MachineName := GVL_const.MachineName,
    StateName := 'AutoMode',
    TimeStamp := GVL_SW.Unix_TimeStamp,
    Value := BOOL_TO_INT(GVL_Visu.AutoMode),
    Enable := tpValueChangeDelay[1].Q); // GenericState
PostHttp[3](
    HostAddress := GVL_const.HttpServerIpAddress,
    HostPort := GVL_const.HttpServerPort,
    ApiEndpoint := GenericState[3].ApiEndpoint,
    JsonPayload := GenericState[3].JsonPayload,
    HttpPostCmd := GenericState[3].HttpPostCmd); // HttpPost
ValueChangeDetector[2](Value := BOOL_TO_INT(GVL_Visu.AutoMode)); // ValueChangeDetector
tpValueChangeDelay[2](IN := ValueChangeDetector[2].ValueChanged, PT := T#50MS); // TP
GenericState[2](
    LineName := GVL_const.LineName,
    MachineName := GVL_const.MachineName,
    StateName := 'DoorOpened',
    TimeStamp := GVL_SW.Unix_TimeStamp,
    Value := BOOL_TO_INT(GVL_Visu.AutoMode),
    Enable := tpValueChangeDelay[2].Q); // GenericState
ValueChangeDetector[3](Value := BOOL_TO_INT(GVL_Visu.LineProducing)); // ValueChangeDetector
tpValueChangeDelay[3](IN := ValueChangeDetector[3].ValueChanged, PT := T#50MS); // TP
GenericState[3](
    LineName := GVL_const.LineName,
    MachineName := GVL_const.MachineName,
    StateName := 'LineProducing',
    TimeStamp := GVL_SW.Unix_TimeStamp,
    Value := BOOL_TO_INT(GVL_Visu.LineProducing),
    Enable := tpValueChangeDelay[3].Q); // GenericState
ValueChangeDetector[4](Value := UINT_TO_INT(GVL_Visu.OkProductCount)); // ValueChangeDetector

END_PROGRAM

// ---- POUs/PRG_10ms/PRG_08_ProductionStatistics.TcPOU
PROGRAM PRG_08_ProductionStatistics
VAR
	PartsPerMinInstant					: PartsPerMinInstant2;
	PartsPerMin							: GenericState;
	PartsPerMinPostHttp					: HttpPost;
	OkPartsPerMinHistorical				: PartsPerMinHistorical;
END_VAR

PartsPerMinInstant(TotalCount := GVL_Visu.OkProductCount); // PartsPerMinInstant2
GVL_Visu.OkPartsPerMinRate := PartsPerMinInstant.PPM;
PartsPerMin(
    LineName := GVL_const.LineName,
    MachineName := GVL_const.MachineName,
    StateName := 'PartsPerMinute',
    TimeStamp := GVL_SW.Unix_TimeStamp,
    Value := TO_INT(PartsPerMinInstant.PPM),
    Enable := GVL_Visu.LineRunning); // GenericState
PartsPerMinPostHttp(
    HostAddress := GVL_const.HttpServerIpAddress,
    HostPort := GVL_const.HttpServerPort,
    ApiEndpoint := PartsPerMin.ApiEndpoint,
    JsonPayload := PartsPerMin.JsonPayload,
    HttpPostCmd := PartsPerMin.HttpPostCmd); // HttpPost
OkPartsPerMinHistorical(ProductSensor := GVL_Visu.SensorProductActive, PartsPerMinHist := GVL_Visu.OkPartsPerMinHistorical); // PartsPerMinHistorical

END_PROGRAM

// ---- POUs/PRG_10ms/PRG_09_PlcDiagnostic.TcPOU
PROGRAM PRG_09_PlcDiagnostic
VAR
	NetID						: 	STRING := '192.168.1.145.1.1';
	tonRecycle50ms				: 	TON;
	tonRecyclePublishMqtt		: 	TON;
	
	CpuMemoryUsage				:	ReadMemoryUsage;
	CpuUsageEx_Core2			:	TC_CPuUsageEx;
	CpuUsageEx_Core3			:	TC_CPuUsageEx;
	CpuLatencyEx_Core2			:	TC_SysLatencyEx;
	CpuLatencyEx_Core3			:	TC_SysLatencyEx;
	
	PlcDiagState				:	ARRAY [1..5] OF GenericState;
	PlcDiagStatePostHttp		:	ARRAY [1..5] OF HttpPost;
END_VAR


// PAGE Recycle Timers for general usage ---
tonRecyclePublishMqtt(IN := NOT tonRecyclePublishMqtt.Q, PT := T#2s); // TON
tonRecycle50ms(IN := NOT tonRecycle50ms.Q, PT := T#50ms); // TON

// PAGE PLC Memory usage ---
CpuMemoryUsage(NetID := NetID); // ReadMemoryUsage
PlcDiagState[1](
    LineName := GVL_const.LineName,
    MachineName := GVL_const.MachineName,
    StateName := GVL_const.PlcCpuMemUsage,
    TimeStamp := GVL_SW.Unix_TimeStamp,
    Value := UINT_TO_INT(CpuMemoryUsage.MemUsage)); // GenericState
PlcDiagStatePostHttp[1](
    HostAddress := GVL_const.HttpServerIpAddress,
    HostPort := GVL_const.HttpServerPort,
    ApiEndpoint := PlcDiagState[1].ApiEndpoint,
    JsonPayload := PlcDiagState[1].JsonPayload,
    HttpPostCmd := PlcDiagState[1].HttpPostCmd); // HttpPost

// PAGE PLC CPU usage ---
CpuUsageEx_Core2(bExecute := tonRecycle50ms.Q, tTimeout := T#5S, sNetId := NetID, nCpuId := 2); // TC_CPuUsageEx
PlcDiagState[2](
    LineName := GVL_const.LineName,
    MachineName := GVL_const.MachineName,
    StateName := GVL_const.PlcCpuCore2Usage,
    TimeStamp := GVL_SW.Unix_TimeStamp,
    Value := UDINT_TO_INT(CpuUsageEx_Core2.nUsage),
    Enable := GVL_Visu.LineRunning AND tonRecyclePublishMqtt.Q); // GenericState
PlcDiagStatePostHttp[2](
    HostAddress := GVL_const.HttpServerIpAddress,
    HostPort := GVL_const.HttpServerPort,
    ApiEndpoint := PlcDiagState[2].ApiEndpoint,
    JsonPayload := PlcDiagState[2].JsonPayload,
    HttpPostCmd := PlcDiagState[2].HttpPostCmd); // HttpPost
CpuUsageEx_Core3(bExecute := tonRecycle50ms.Q, tTimeout := T#5S, sNetId := NetID, nCpuId := 3); // TC_CPuUsageEx
PlcDiagState[3](
    LineName := GVL_const.LineName,
    MachineName := GVL_const.MachineName,
    StateName := GVL_const.PlcCpuCore3Usage,
    TimeStamp := GVL_SW.Unix_TimeStamp,
    Value := UDINT_TO_INT(CpuUsageEx_Core3.nUsage),
    Enable := GVL_Visu.LineRunning AND tonRecyclePublishMqtt.Q); // GenericState
PlcDiagStatePostHttp[3](
    HostAddress := GVL_const.HttpServerIpAddress,
    HostPort := GVL_const.HttpServerPort,
    ApiEndpoint := PlcDiagState[3].ApiEndpoint,
    JsonPayload := PlcDiagState[3].JsonPayload,
    HttpPostCmd := PlcDiagState[3].HttpPostCmd); // HttpPost

// PAGE PLC CPU latency
CpuLatencyEx_Core2(bExecute := tonRecycle50ms.Q, tTimeout := T#5S, sNetId := NetID, nCpuId := 2); // TC_SysLatencyEx
PlcDiagState[4](
    LineName := GVL_const.LineName,
    MachineName := GVL_const.MachineName,
    StateName := GVL_const.PlcCpuCore2Jitter,
    TimeStamp := GVL_SW.Unix_TimeStamp,
    Value := UDINT_TO_INT(CpuLatencyEx_Core2.nActual),
    Enable := GVL_Visu.LineRunning AND tonRecyclePublishMqtt.Q); // GenericState
PlcDiagStatePostHttp[4](
    HostAddress := GVL_const.HttpServerIpAddress,
    HostPort := GVL_const.HttpServerPort,
    ApiEndpoint := PlcDiagState[4].ApiEndpoint,
    JsonPayload := PlcDiagState[4].JsonPayload,
    HttpPostCmd := PlcDiagState[4].HttpPostCmd); // HttpPost
CpuLatencyEx_Core3(bExecute := tonRecycle50ms.Q, tTimeout := T#5S, sNetId := NetID, nCpuId := 3); // TC_SysLatencyEx
PlcDiagState[5](
    LineName := GVL_const.LineName,
    MachineName := GVL_const.MachineName,
    StateName := GVL_const.PlcCpuCore3Jitter,
    TimeStamp := GVL_SW.Unix_TimeStamp,
    Value := UDINT_TO_INT(CpuLatencyEx_Core3.nActual),
    Enable := GVL_Visu.LineRunning AND tonRecyclePublishMqtt.Q); // GenericState
PlcDiagStatePostHttp[5](
    HostAddress := GVL_const.HttpServerIpAddress,
    HostPort := GVL_const.HttpServerPort,
    ApiEndpoint := PlcDiagState[5].ApiEndpoint,
    JsonPayload := PlcDiagState[5].JsonPayload,
    HttpPostCmd := PlcDiagState[5].HttpPostCmd); // HttpPost
// GVL_Visu.LineRunning AND tonRecyclePublishMqtt.Q: input not connected

END_PROGRAM

// ---- POUs/PRG_10ms/PRG_13_MES.TcPOU
PROGRAM PRG_13_MES
VAR
	MesData					: HttpGet;
	tonRecycle01			: TON;
END_VAR

tonRecycle01(IN := NOT tonRecycle01.Q, PT := T#2S); // TON
MesData(
    HostAddress := GVL_const.HttpServerIpAddress,
    HostPort := GVL_const.HttpServerPort,
    ApiEndpoint := '/production_orders',
    HttpGetCmd := tonRecycle01.Q); // HttpGet

END_PROGRAM

// ---- POUs/PRG_10ms/PRG_11_AirFlowAnalytics.TcPOU
PROGRAM PRG_11_AirFlowAnalytics
VAR
	AirFlowRateSensor: GenericSensor;
	AirPressureSensor: GenericSensor;
	AirTemperatureSensor: GenericSensor;
	
	AirFlowSensorPostHttp: HttpPost;
	AirPresSensorPostHttp: HttpPost;
	AirTempSensorPostHttp: HttpPost;
END_VAR

AirFlowRateSensor(
    LineName := GVL_const.LineName,
    MachineName := GVL_const.MachineName,
    SensorName := GVL_const.AirFlowSensor,
    TimeStamp := GVL_SW.Unix_TimeStamp,
    Value := GVL_Visu.AirFlowRate,
    Enable := GVL_Visu.LineRunning); // GenericSensor
AirFlowSensorPostHttp(
    HostAddress := GVL_const.HttpServerIpAddress,
    HostPort := GVL_const.HttpServerPort,
    ApiEndpoint := AirFlowRateSensor.ApiEndpoint,
    JsonPayload := AirFlowRateSensor.JsonPayload,
    HttpPostCmd := AirFlowRateSensor.HttpPostCmd); // HttpPost
AirPressureSensor(
    LineName := GVL_const.LineName,
    MachineName := GVL_const.MachineName,
    SensorName := GVL_const.AirPresSensor,
    TimeStamp := GVL_SW.Unix_TimeStamp,
    Value := GVL_Visu.AirPressure,
    Enable := GVL_Visu.LineRunning); // GenericSensor
AirPresSensorPostHttp(
    HostAddress := GVL_const.HttpServerIpAddress,
    HostPort := GVL_const.HttpServerPort,
    ApiEndpoint := AirPressureSensor.ApiEndpoint,
    JsonPayload := AirPressureSensor.JsonPayload,
    HttpPostCmd := AirPressureSensor.HttpPostCmd); // HttpPost
AirTemperatureSensor(
    LineName := GVL_const.LineName,
    MachineName := GVL_const.MachineName,
    SensorName := GVL_const.AirTempSensor,
    TimeStamp := GVL_SW.Unix_TimeStamp,
    Value := GVL_Visu.AirTemperature,
    Enable := GVL_Visu.LineRunning); // GenericSensor
AirTempSensorPostHttp(
    HostAddress := GVL_const.HttpServerIpAddress,
    HostPort := GVL_const.HttpServerPort,
    ApiEndpoint := AirTemperatureSensor.ApiEndpoint,
    JsonPayload := AirTemperatureSensor.JsonPayload,
    HttpPostCmd := AirTemperatureSensor.HttpPostCmd); // HttpPost
// GVL_SW.AirVolumetricFlowRate: input not connected
// GVL_SW.AirPressure: input not connected
// GVL_SW.AirTemperature: input not connected

END_PROGRAM

// ---- POUs/PRG_10ms/PRG_10_TempHumidAnalytics.TcPOU
PROGRAM PRG_10_TempHumidAnalytics
VAR
	TempSensor								: GenericSensor;
	HumiditySensor							: GenericSensor;
	
	TempSensorPostHTTP						: HttpPost;
	HumiditySensorPostHTTP					: HttpPost;
END_VAR

TempSensor(
    LineName := GVL_const.LineName,
    MachineName := GVL_const.MachineName,
    SensorName := GVL_const.AmbientTempSensor,
    TimeStamp := GVL_SW.Unix_TimeStamp,
    Value := GVL_Visu.AmbientTemperature,
    Enable := GVL_Visu.LineRunning); // GenericSensor
TempSensorPostHTTP(
    HostAddress := GVL_const.HttpServerIpAddress,
    HostPort := GVL_const.HttpServerPort,
    ApiEndpoint := TempSensor.ApiEndpoint,
    JsonPayload := TempSensor.JsonPayload,
    HttpPostCmd := TempSensor.HttpPostCmd); // HttpPost
HumiditySensor(
    LineName := GVL_const.LineName,
    MachineName := GVL_const.MachineName,
    SensorName := GVL_const.AmbientHumiditySensor,
    TimeStamp := GVL_SW.Unix_TimeStamp,
    Value := GVL_Visu.AmbientHumidity,
    Enable := GVL_Visu.LineRunning); // GenericSensor
HumiditySensorPostHTTP(
    HostAddress := GVL_const.HttpServerIpAddress,
    HostPort := GVL_const.HttpServerPort,
    ApiEndpoint := HumiditySensor.ApiEndpoint,
    JsonPayload := HumiditySensor.JsonPayload,
    HttpPostCmd := HumiditySensor.HttpPostCmd); // HttpPost
// GVL_SW.AmbientTempSensor: input not connected
// GVL_SW.AmbientHumiditySensor: input not connected

END_PROGRAM

// ---- POUs/PRG_10ms/PRG_12_OilContaminationAnalytics.TcPOU
PROGRAM PRG_12_OilContaminationAnalytics
VAR
	OilDiffPressSensor: GenericSensor;
	OilDiffPressSensorPostHttp: HttpPost;
END_VAR

OilDiffPressSensor(
    LineName := GVL_const.LineName,
    MachineName := GVL_const.MachineName,
    SensorName := GVL_const.DiffPressSensor1,
    TimeStamp := GVL_SW.Unix_TimeStamp,
    Value := GVL_Visu.OilDiffPressure,
    Enable := GVL_Visu.LineRunning); // GenericSensor
OilDiffPressSensorPostHttp(
    HostAddress := GVL_const.HttpServerIpAddress,
    HostPort := GVL_const.HttpServerPort,
    ApiEndpoint := OilDiffPressSensor.ApiEndpoint,
    JsonPayload := OilDiffPressSensor.JsonPayload,
    HttpPostCmd := OilDiffPressSensor.HttpPostCmd); // HttpPost
// GVL_SW.DiffPressSensor: input not connected

END_PROGRAM
